C03569=1015.832,-110.510,-100.414,164.984,56.890,160.011
C03570=1015.836,-110.261,-100.421,164.987,56.884,160.010
C03571=1015.842,-110.011,-100.428,164.990,56.879,160.010
C03572=1015.846,-109.761,-100.435,164.993,56.872,160.010
C03573=1015.852,-109.511,-100.444,164.995,56.866,160.009
C03574=1015.857,-109.261,-100.452,164.999,56.860,160.009
C03575=1015.861,-109.012,-100.460,165.001,56.854,160.009
C03576=1015.866,-108.762,-100.468,165.003,56.847,160.008
C03577=1015.871,-108.511,-100.475,165.007,56.841,160.008
C03578=1015.876,-108.262,-100.484,165.010,56.835,160.007
C03579=1015.881,-108.012,-100.491,165.013,56.829,160.007
C03580=1015.886,-107.762,-100.499,165.016,56.823,160.007
C03581=1015.890,-107.513,-100.507,165.018,56.817,160.006
C03582=1015.895,-107.262,-100.515,165.022,56.811,160.006
C03583=1015.901,-107.013,-100.523,165.024,56.805,160.006
C03584=1015.905,-106.763,-100.531,165.027,56.799,160.005
C03585=1015.910,-106.513,-100.539,165.030,56.793,160.005
C03586=1015.915,-106.263,-100.547,165.033,56.787,160.005
C03587=1015.920,-106.014,-100.555,165.036,56.780,160.004
C03588=1015.925,-105.764,-100.563,165.039,56.774,160.004
C03589=1015.930,-105.514,-100.571,165.041,56.769,160.003
C03590=1015.934,-105.264,-100.579,165.045,56.762,160.003
C03591=1015.940,-105.014,-100.587,165.047,56.757,160.003
C03592=1015.945,-104.765,-100.596,165.051,56.750,160.003
C03593=1015.950,-104.514,-100.604,165.053,56.744,160.002
C03594=1015.955,-104.265,-100.612,165.056,56.738,160.002
C03595=1015.959,-104.015,-100.619,165.059,56.732,160.001
C03596=1015.965,-103.765,-100.628,165.062,56.726,160.001
C03597=1015.970,-103.515,-100.636,165.066,56.720,160.001
C03598=1015.974,-103.266,-100.644,165.068,56.713,160.000
C03599=1015.979,-103.016,-100.653,165.070,56.708,160.000
C03600=1015.984,-102.766,-100.661,165.074,56.701,160.000
C03601=1015.989,-102.516,-100.669,165.077,56.696,159.999
C03602=1015.995,-102.234,-100.678,165.080,56.689,159.999
C03603=1016.000,-101.952,-100.688,165.083,56.682,159.998
C03604=1016.006,-101.669,-100.697,165.087,56.674,159.998
C03605=1016.011,-101.387,-100.706,165.090,56.667,159.998
C03606=1016.016,-101.138,-100.715,165.093,56.662,159.997
C03607=1016.021,-100.887,-100.722,165.096,56.655,159.997
C03608=1016.027,-100.638,-100.731,165.098,56.649,159.996
C03609=1016.032,-100.388,-100.739,165.102,56.643,159.996
C03610=1016.037,-100.139,-100.747,165.104,56.636,159.996
C03611=1016.042,-99.888,-100.755,165.107,56.630,159.995
C03612=1016.046,-99.638,-100.764,165.110,56.624,159.995
C03613=1016.051,-99.389,-100.773,165.112,56.618,159.994
C03614=1016.057,-99.139,-100.781,165.116,56.612,159.994
C03615=1016.062,-98.889,-100.789,165.119,56.606,159.994
C03616=1016.066,-98.640,-100.797,165.122,56.599,159.993
C03617=1016.071,-98.390,-100.806,165.124,56.593,159.993
C03618=1016.077,-98.140,-100.814,165.128,56.587,159.993
C03619=1016.082,-97.890,-100.822,165.130,56.580,159.992
C03620=1016.086,-97.640,-100.831,165.134,56.574,159.992
C03621=1016.091,-97.390,-100.839,165.136,56.569,159.991
C03622=1016.096,-97.140,-100.849,165.139,56.563,159.991
C03623=1016.101,-96.890,-100.857,165.143,56.557,159.991
C03624=1016.107,-96.641,-100.865,165.145,56.551,159.990
C03625=1016.111,-96.391,-100.875,165.147,56.544,159.990
C03626=1016.116,-96.141,-100.883,165.151,56.538,159.990
C03627=1016.120,-95.892,-100.892,165.154,56.532,159.989
C03628=1016.126,-95.642,-100.900,165.157,56.526,159.989
C03629=1016.131,-95.392,-100.909,165.160,56.520,159.989
C03630=1016.135,-95.142,-100.918,165.162,56.514,159.988
C03631=1016.141,-94.892,-100.926,165.166,56.508,159.988
C03632=1016.146,-94.643,-100.935,165.168,56.502,159.987
C03633=1016.150,-94.393,-100.944,165.172,56.496,159.987
C03634=1016.156,-94.143,-100.952,165.174,56.489,159.987
C03635=1016.160,-93.893,-100.961,165.177,56.484,159.986
C03636=1016.165,-93.643,-100.970,165.180,56.477,159.986
C03637=1016.171,-93.394,-100.978,165.183,56.472,159.986
C03638=1016.175,-93.144,-100.987,165.186,56.465,159.985
C03639=1016.180,-92.894,-100.996,165.189,56.459,159.985
C03640=1016.185,-92.644,-101.005,165.192,56.453,159.985
C03641=1016.190,-92.394,-101.014,165.194,56.446,159.984
C03642=1016.196,-92.144,-101.022,165.197,56.441,159.983
C03643=1016.200,-91.894,-101.031,165.201,56.434,159.983
C03644=1016.206,-91.645,-101.040,165.203,56.428,159.983
C03645=1016.210,-91.395,-101.049,165.206,56.422,159.982
C03646=1016.215,-91.145,-101.058,165.209,56.416,159.982
C03647=1016.221,-90.896,-101.066,165.212,56.409,159.982
C03648=1016.225,-90.646,-101.075,165.215,56.403,159.981
C03649=1016.230,-90.396,-101.084,165.218,56.397,159.981
C03650=1016.235,-90.146,-101.093,165.221,56.391,159.980
C03651=1016.240,-89.896,-101.101,165.224,56.385,159.980
C03652=1016.246,-89.647,-101.111,165.227,56.379,159.980
C03653=1016.250,-89.397,-101.120,165.230,56.372,159.979
C03654=1016.256,-89.147,-101.128,165.233,56.366,159.979
C03655=1016.260,-88.897,-101.137,165.236,56.359,159.978
C03656=1016.266,-88.647,-101.146,165.238,56.354,159.978
C03657=1016.272,-88.398,-101.155,165.242,56.347,159.978
C03658=1016.276,-88.148,-101.164,165.244,56.341,159.977
C03659=1016.281,-87.898,-101.173,165.248,56.335,159.977
C03660=1016.286,-87.648,-101.182,165.250,56.328,159.976
C03661=1016.291,-87.398,-101.191,165.254,56.322,159.976
C03662=1016.296,-87.149,-101.200,165.256,56.316,159.975
C03663=1016.301,-86.899,-101.209,165.259,56.309,159.975
C03664=1016.307,-86.650,-101.217,165.261,56.303,159.975
C03665=1016.312,-86.399,-101.227,165.265,56.297,159.974
C03666=1016.317,-86.120,-101.237,165.268,56.290,159.974
C03667=1016.324,-85.839,-101.247,165.271,56.283,159.973
C03668=1016.329,-85.559,-101.257,165.274,56.275,159.973
C03669=1016.334,-85.278,-101.267,165.278,56.268,159.972
C03670=1016.340,-85.029,-101.276,165.281,56.262,159.972
C03671=1016.345,-84.779,-101.286,165.284,56.256,159.972
C03672=1016.350,-84.530,-101.294,165.287,56.250,159.971
C03673=1016.355,-84.280,-101.303,165.290,56.243,159.971
C03674=1016.361,-84.030,-101.313,165.293,56.237,159.970
C03675=1016.366,-83.780,-101.321,165.296,56.230,159.970
C03676=1016.370,-83.530,-101.330,165.298,56.224,159.969
C03677=1016.376,-83.281,-101.339,165.301,56.218,159.969
C03678=1016.381,-83.031,-101.348,165.305,56.211,159.969
C03679=1016.386,-82.780,-101.357,165.307,56.205,159.968
C03680=1016.392,-82.531,-101.367,165.310,56.198,159.968
C03681=1016.396,-82.281,-101.376,165.313,56.193,159.967
C03682=1016.402,-82.032,-101.385,165.316,56.186,159.967
C03683=1016.407,-81.782,-101.394,165.319,56.179,159.966
C03684=1016.412,-81.532,-101.403,165.322,56.173,159.966
C03685=1016.417,-81.282,-101.413,165.325,56.166,159.965
C03686=1016.422,-81.033,-101.421,165.328,56.160,159.965
C03687=1016.429,-80.783,-101.431,165.331,56.154,159.965
C03688=1016.433,-80.533,-101.440,165.334,56.147,159.964
C03689=1016.438,-80.283,-101.448,165.337,56.141,159.964
C03690=1016.443,-80.034,-101.458,165.340,56.134,159.963
C03691=1016.449,-79.784,-101.468,165.343,56.128,159.963
C03692=1016.454,-79.534,-101.477,165.346,56.122,159.962
C03693=1016.459,-79.285,-101.486,165.348,56.116,159.962
C03694=1016.464,-79.034,-101.496,165.352,56.109,159.962
C03695=1016.469,-78.784,-101.506,165.354,56.103,159.961
C03696=1016.474,-78.535,-101.515,165.357,56.096,159.961
C03697=1016.479,-78.285,-101.524,165.360,56.091,159.960
C03698=1016.484,-78.035,-101.534,165.364,56.085,159.960
C03699=1016.490,-77.786,-101.543,165.366,56.078,159.959
C03700=1016.494,-77.536,-101.552,165.370,56.072,159.959
C03701=1016.500,-77.286,-101.563,165.372,56.066,159.959
C03702=1016.505,-77.037,-101.572,165.375,56.059,159.958
C03703=1016.510,-76.787,-101.581,165.378,56.053,159.958
C03704=1016.515,-76.537,-101.591,165.381,56.046,159.957
C03705=1016.520,-76.287,-101.601,165.383,56.040,159.957
C03706=1016.525,-76.038,-101.609,165.387,56.034,159.956
C03707=1016.531,-75.787,-101.619,165.389,56.028,159.956
C03708=1016.536,-75.538,-101.629,165.392,56.021,159.955
C03709=1016.541,-75.287,-101.639,165.395,56.015,159.955
C03710=1016.546,-75.038,-101.648,165.398,56.008,159.955
C03711=1016.551,-74.789,-101.658,165.401,56.003,159.954
C03712=1016.557,-74.539,-101.668,165.404,55.996,159.954
C03713=1016.561,-74.289,-101.677,165.407,55.990,159.953
C03714=1016.567,-74.039,-101.687,165.410,55.983,159.953
C03715=1016.571,-73.789,-101.697,165.413,55.978,159.952
C03716=1016.576,-73.540,-101.707,165.416,55.972,159.952
C03717=1016.582,-73.290,-101.717,165.418,55.965,159.952
C03718=1016.587,-73.040,-101.727,165.421,55.959,159.951
C03719=1016.592,-72.790,-101.737,165.424,55.953,159.951
C03720=1016.597,-72.541,-101.747,165.427,55.947,159.950
C03721=1016.602,-72.291,-101.757,165.431,55.941,159.950
C03722=1016.607,-72.041,-101.767,165.433,55.934,159.949
C03723=1016.612,-71.792,-101.776,165.436,55.929,159.949
C03724=1016.617,-71.542,-101.787,165.439,55.922,159.949
C03725=1016.622,-71.292,-101.796,165.441,55.916,159.948
C03726=1016.628,-71.042,-101.806,165.445,55.910,159.948
C03727=1016.632,-70.793,-101.816,165.447,55.904,159.947
C03728=1016.638,-70.543,-101.826,165.451,55.897,159.947
C03729=1016.643,-70.293,-101.836,165.453,55.891,159.946
C03730=1016.649,-70.015,-101.847,165.456,55.884,159.946
C03731=1016.654,-69.737,-101.859,165.460,55.877,159.945
C03732=1016.660,-69.458,-101.870,165.463,55.870,159.945
C03733=1016.665,-69.180,-101.880,165.466,55.864,159.944
C03734=1016.671,-68.930,-101.890,165.469,55.857,159.944
C03735=1016.676,-68.681,-101.900,165.472,55.851,159.944
C03736=1016.681,-68.430,-101.910,165.475,55.844,159.943
C03737=1016.686,-68.181,-101.920,165.478,55.839,159.943
C03738=1016.692,-67.932,-101.931,165.481,55.832,159.942
C03739=1016.697,-67.681,-101.941,165.484,55.826,159.942
C03740=1016.702,-67.432,-101.951,165.487,55.819,159.941
C03741=1016.707,-67.182,-101.961,165.489,55.814,159.941
C03742=1016.712,-66.933,-101.971,165.493,55.807,159.941
C03743=1016.717,-66.682,-101.982,165.495,55.801,159.940
C03744=1016.722,-66.433,-101.992,165.499,55.794,159.940
C03745=1016.727,-66.183,-102.002,165.501,55.788,159.939
C03746=1016.732,-65.933,-102.012,165.504,55.782,159.939
C03747=1016.738,-65.684,-102.022,165.507,55.775,159.938
C03748=1016.743,-65.434,-102.033,165.510,55.769,159.938
C03749=1016.748,-65.184,-102.042,165.512,55.763,159.937
C03750=1016.753,-64.934,-102.053,165.516,55.756,159.937
C03751=1016.758,-64.685,-102.062,165.518,55.750,159.936
C03752=1016.764,-64.435,-102.072,165.522,55.744,159.936
C03753=1016.769,-64.185,-102.083,165.524,55.738,159.935
C03754=1016.774,-63.936,-102.093,165.527,55.731,159.935
C03755=1016.780,-63.686,-102.103,165.530,55.725,159.934
C03756=1016.784,-63.436,-102.113,165.533,55.719,159.934
C03757=1016.790,-63.186,-102.123,165.537,55.712,159.934
C03758=1016.796,-62.937,-102.134,165.539,55.705,159.933
C03759=1016.800,-62.687,-102.144,165.543,55.699,159.933
C03760=1016.806,-62.437,-102.154,165.545,55.693,159.932
C03761=1016.811,-62.187,-102.164,165.548,55.686,159.932
C03762=1016.816,-61.938,-102.175,165.551,55.680,159.931
C03763=1016.822,-61.688,-102.185,165.554,55.674,159.931
C03764=1016.827,-61.438,-102.195,165.556,55.667,159.930
C03765=1016.831,-61.188,-102.205,165.560,55.661,159.930
C03766=1016.837,-60.939,-102.216,165.562,55.655,159.929
C03767=1016.843,-60.689,-102.227,165.565,55.648,159.929
C03768=1016.847,-60.439,-102.236,165.568,55.641,159.928
C03769=1016.853,-60.190,-102.247,165.571,55.635,159.928
C03770=1016.859,-59.940,-102.257,165.574,55.629,159.927
C03771=1016.863,-59.690,-102.267,165.576,55.622,159.927
C03772=1016.869,-59.440,-102.277,165.580,55.615,159.926
C03773=1016.875,-59.191,-102.288,165.582,55.610,159.926
C03774=1016.880,-58.940,-102.298,165.586,55.603,159.925
C03775=1016.885,-58.691,-102.308,165.589,55.596,159.925
C03776=1016.891,-58.442,-102.319,165.591,55.590,159.924
C03777=1016.896,-58.191,-102.329,165.595,55.584,159.924
C03778=1016.902,-57.942,-102.340,165.597,55.577,159.923
C03779=1016.907,-57.693,-102.350,165.600,55.570,159.923
C03780=1016.912,-57.442,-102.360,165.603,55.564,159.922
C03781=1016.918,-57.193,-102.371,165.606,55.557,159.922
C03782=1016.922,-56.943,-102.382,165.609,55.550,159.921
C03783=1016.928,-56.694,-102.392,165.612,55.545,159.921
C03784=1016.933,-56.444,-102.402,165.615,55.538,159.920
C03785=1016.938,-56.194,-102.412,165.618,55.531,159.920
C03786=1016.944,-55.944,-102.423,165.620,55.525,159.919
C03787=1016.950,-55.694,-102.434,165.623,55.518,159.919
C03788=1016.955,-55.445,-102.444,165.626,55.512,159.918
C03789=1016.960,-55.195,-102.454,165.629,55.506,159.918
C03790=1016.966,-54.946,-102.465,165.633,55.499,159.917
C03791=1016.971,-54.695,-102.475,165.635,55.492,159.917
C03792=1016.977,-54.445,-102.485,165.638,55.486,159.916
C03793=1016.982,-54.197,-102.496,165.640,55.479,159.915
C03794=1016.988,-53.919,-102.508,165.644,55.471,159.915
C03795=1016.995,-53.642,-102.520,165.647,55.465,159.914
C03796=1017.000,-53.365,-102.531,165.650,55.457,159.914
C03797=1017.006,-53.088,-102.543,165.654,55.450,159.913
C03798=1017.012,-52.838,-102.553,165.657,55.444,159.913
C03799=1017.017,-52.588,-102.564,165.660,55.437,159.912
C03800=1017.022,-52.338,-102.575,165.662,55.430,159.912
C03801=1017.027,-52.089,-102.585,165.665,55.424,159.911
C03802=1017.033,-51.839,-102.596,165.668,55.417,159.911
C03803=1017.038,-51.589,-102.606,165.671,55.410,159.910
C03804=1017.044,-51.340,-102.617,165.674,55.404,159.909
C03805=1017.050,-51.090,-102.627,165.677,55.397,159.909
C03806=1017.055,-50.840,-102.638,165.679,55.391,159.908
///RCONF 1,0,0,0,0,0,0,0,0,0,0,0,0,0,0,0,0,0,0,0,0,0,0,0
C03807=1017.060,-50.590,-102.649,165.683,55.384,159.908
C03808=1017.065,-50.340,-102.661,165.685,55.378,159.907
C03809=1017.071,-50.090,-102.671,165.689,55.371,159.907
C03810=1017.076,-49.841,-102.682,165.691,55.366,159.906
C03811=1017.081,-49.591,-102.693,165.695,55.359,159.906
C03812=1017.086,-49.341,-102.705,165.697,55.353,159.905
C03813=1017.092,-49.091,-102.715,165.701,55.347,159.905
C03814=1017.097,-48.842,-102.725,165.703,55.340,159.904
C03815=1017.102,-48.593,-102.737,165.705,55.334,159.904
C03816=1017.108,-48.343,-102.748,165.708,55.327,159.903
C03817=1017.113,-48.093,-102.759,165.711,55.321,159.903
C03818=1017.119,-47.844,-102.770,165.714,55.315,159.902
C03819=1017.123,-47.593,-102.781,165.716,55.308,159.902
C03820=1017.129,-47.344,-102.792,165.720,55.302,159.901
C03821=1017.134,-47.094,-102.803,165.722,55.296,159.901
C03822=1017.140,-46.845,-102.814,165.726,55.289,159.900
C03823=1017.145,-46.595,-102.826,165.728,55.283,159.900
C03824=1017.150,-46.345,-102.837,165.731,55.276,159.899
C03825=1017.155,-46.095,-102.848,165.734,55.270,159.899
C03826=1017.161,-45.846,-102.859,165.737,55.264,159.898
C03827=1017.166,-45.596,-102.870,165.739,55.257,159.898
C03828=1017.172,-45.347,-102.881,165.743,55.251,159.897
C03829=1017.177,-45.096,-102.892,165.746,55.244,159.897
C03830=1017.182,-44.847,-102.903,165.749,55.238,159.896
C03831=1017.187,-44.597,-102.914,165.752,55.231,159.896
C03832=1017.193,-44.347,-102.925,165.754,55.225,159.895
C03833=1017.198,-44.098,-102.937,165.757,55.218,159.895
C03834=1017.204,-43.848,-102.948,165.760,55.212,159.894
C03835=1017.209,-43.598,-102.959,165.763,55.205,159.893
C03836=1017.215,-43.349,-102.970,165.765,55.199,159.893
C03837=1017.220,-43.099,-102.981,165.769,55.193,159.893
C03838=1017.225,-42.850,-102.992,165.771,55.186,159.892
C03839=1017.230,-42.600,-103.004,165.775,55.180,159.891
C03840=1017.236,-42.350,-103.015,165.777,55.173,159.891
C03841=1017.241,-42.101,-103.026,165.780,55.167,159.890
C03842=1017.247,-41.850,-103.037,165.782,55.160,159.890
C03843=1017.252,-41.601,-103.049,165.786,55.154,159.889
C03844=1017.258,-41.351,-103.060,165.789,55.147,159.889
C03845=1017.263,-41.101,-103.071,165.791,55.140,159.888
C03846=1017.269,-40.852,-103.082,165.794,55.134,159.887
C03847=1017.274,-40.602,-103.093,165.797,55.128,159.887
C03848=1017.280,-40.352,-103.104,165.800,55.121,159.887
C03849=1017.285,-40.103,-103.116,165.803,55.115,159.886
C03850=1017.291,-39.854,-103.127,165.806,55.108,159.885
C03851=1017.296,-39.604,-103.139,165.809,55.102,159.885
C03852=1017.301,-39.353,-103.151,165.811,55.095,159.884
C03853=1017.307,-39.104,-103.162,165.815,55.088,159.884
C03854=1017.312,-38.854,-103.173,165.817,55.082,159.883
C03855=1017.317,-38.604,-103.185,165.820,55.077,159.883
C03856=1017.322,-38.355,-103.197,165.823,55.070,159.882
C03857=1017.328,-38.106,-103.208,165.825,55.063,159.881
C03858=1017.334,-37.828,-103.221,165.829,55.057,159.881
C03859=1017.339,-37.551,-103.233,165.831,55.049,159.880
C03860=1017.346,-37.275,-103.246,165.835,55.043,159.880
C03861=1017.351,-36.998,-103.259,165.838,55.035,159.879
C03862=1017.356,-36.748,-103.270,165.841,55.028,159.879
C03863=1017.362,-36.499,-103.283,165.843,55.023,159.878
C03864=1017.368,-36.249,-103.294,165.847,55.016,159.878
C03865=1017.373,-35.999,-103.305,165.849,55.010,159.877
C03866=1017.378,-35.750,-103.318,165.852,55.003,159.876
C03867=1017.383,-35.500,-103.329,165.855,54.997,159.876
C03868=1017.389,-35.250,-103.341,165.858,54.990,159.875
C03869=1017.395,-35.001,-103.352,165.860,54.984,159.875
C03870=1017.400,-34.751,-103.364,165.864,54.978,159.874
C03871=1017.405,-34.501,-103.375,165.866,54.971,159.874
C03872=1017.410,-34.252,-103.388,165.870,54.965,159.873
C03873=1017.416,-34.002,-103.399,165.872,54.958,159.873
C03874=1017.422,-33.752,-103.410,165.875,54.952,159.872
C03875=1017.427,-33.503,-103.422,165.877,54.945,159.871
C03876=1017.432,-33.253,-103.434,165.881,54.939,159.871
C03877=1017.438,-33.003,-103.446,165.883,54.932,159.870
C03878=1017.443,-32.753,-103.458,165.886,54.925,159.870
C03879=1017.449,-32.504,-103.469,165.888,54.919,159.869
C03880=1017.454,-32.255,-103.481,165.892,54.912,159.869
C03881=1017.459,-32.004,-103.493,165.895,54.907,159.868
C03882=1017.465,-31.755,-103.505,165.898,54.900,159.868
C03883=1017.470,-31.505,-103.517,165.900,54.894,159.867
C03884=1017.476,-31.256,-103.528,165.903,54.887,159.867
C03885=1017.481,-31.006,-103.540,165.906,54.881,159.866
C03886=1017.486,-30.756,-103.551,165.909,54.874,159.865
C03887=1017.492,-30.507,-103.564,165.911,54.868,159.865
C03888=1017.497,-30.256,-103.575,165.915,54.861,159.864
C03889=1017.503,-30.008,-103.587,165.917,54.855,159.864
C03890=1017.508,-29.758,-103.599,165.920,54.848,159.863
C03891=1017.514,-29.508,-103.611,165.923,54.842,159.862
C03892=1017.519,-29.258,-103.623,165.926,54.835,159.862
C03893=1017.525,-29.009,-103.635,165.928,54.829,159.861
C03894=1017.531,-28.759,-103.646,165.931,54.822,159.861
C03895=1017.536,-28.510,-103.658,165.935,54.815,159.860
C03896=1017.541,-28.260,-103.670,165.937,54.809,159.860
C03897=1017.547,-28.010,-103.682,165.940,54.802,159.859
C03898=1017.552,-27.760,-103.694,165.942,54.795,159.858
C03899=1017.557,-27.511,-103.706,165.946,54.789,159.858
C03900=1017.563,-27.261,-103.718,165.948,54.783,159.857
C03901=1017.568,-27.011,-103.730,165.951,54.777,159.857
C03902=1017.574,-26.762,-103.742,165.954,54.770,159.856
C03903=1017.580,-26.512,-103.755,165.956,54.764,159.855
C03904=1017.585,-26.262,-103.766,165.959,54.757,159.855
C03905=1017.591,-26.012,-103.779,165.962,54.751,159.854
C03906=1017.596,-25.763,-103.791,165.965,54.744,159.854
C03907=1017.601,-25.514,-103.803,165.968,54.739,159.853
C03908=1017.607,-25.264,-103.815,165.970,54.732,159.853
C03909=1017.611,-25.014,-103.828,165.973,54.726,159.852
C03910=1017.617,-24.764,-103.840,165.976,54.719,159.852
C03911=1017.623,-24.515,-103.852,165.979,54.713,159.851
C03912=1017.628,-24.265,-103.864,165.981,54.706,159.850
C03913=1017.633,-24.015,-103.876,165.985,54.700,159.850
C03914=1017.639,-23.766,-103.889,165.987,54.693,159.849
C03915=1017.645,-23.516,-103.901,165.989,54.687,159.849
C03916=1017.650,-23.266,-103.913,165.993,54.680,159.848
C03917=1017.655,-23.017,-103.925,165.995,54.674,159.847
C03918=1017.661,-22.767,-103.937,165.998,54.667,159.847
C03919=1017.666,-22.518,-103.950,166.001,54.661,159.846
C03920=1017.671,-22.268,-103.963,166.004,54.654,159.846
C03921=1017.676,-22.018,-103.974,166.006,54.648,159.845
C03922=1017.683,-21.741,-103.988,166.010,54.641,159.845
C03923=1017.689,-21.463,-104.001,166.012,54.634,159.844
C03924=1017.695,-21.185,-104.015,166.015,54.627,159.843
C03925=1017.701,-20.907,-104.029,166.019,54.620,159.843
C03926=1017.707,-20.658,-104.041,166.022,54.613,159.842
C03927=1017.713,-20.408,-104.054,166.024,54.606,159.841
C03928=1017.718,-20.158,-104.065,166.027,54.600,159.841
C03929=1017.724,-19.908,-104.078,166.029,54.593,159.840
C03930=1017.728,-19.659,-104.091,166.033,54.587,159.840
C03931=1017.734,-19.409,-104.103,166.035,54.580,159.839
C03932=1017.739,-19.160,-104.116,166.038,54.574,159.838
C03933=1017.745,-18.910,-104.128,166.041,54.567,159.838
C03934=1017.751,-18.661,-104.140,166.044,54.561,159.837
C03935=1017.756,-18.411,-104.153,166.046,54.555,159.837
C03936=1017.762,-18.162,-104.165,166.050,54.548,159.836
C03937=1017.768,-17.912,-104.178,166.052,54.542,159.835
C03938=1017.773,-17.663,-104.190,166.055,54.535,159.835
C03939=1017.778,-17.412,-104.202,166.058,54.529,159.834
C03940=1017.783,-17.163,-104.214,166.061,54.522,159.834
C03941=1017.789,-16.913,-104.227,166.063,54.515,159.833
C03942=1017.795,-16.663,-104.240,166.066,54.508,159.832
C03943=1017.800,-16.414,-104.252,166.069,54.502,159.832
C03944=1017.806,-16.164,-104.264,166.072,54.495,159.831
C03945=1017.811,-15.915,-104.276,166.074,54.489,159.830
C03946=1017.817,-15.665,-104.290,166.078,54.482,159.830
C03947=1017.822,-15.416,-104.302,166.080,54.476,159.829
C03948=1017.828,-15.166,-104.315,166.082,54.470,159.829
C03949=1017.833,-14.917,-104.328,166.086,54.463,159.828
C03950=1017.839,-14.667,-104.340,166.088,54.457,159.827
C03951=1017.844,-14.417,-104.354,166.090,54.451,159.827
C03952=1017.849,-14.167,-104.366,166.094,54.444,159.826
C03953=1017.855,-13.917,-104.378,166.096,54.438,159.826
C03954=1017.860,-13.669,-104.392,166.099,54.431,159.825
C03955=1017.866,-13.419,-104.404,166.102,54.425,159.824
C03956=1017.871,-13.168,-104.417,166.104,54.419,159.824
C03957=1017.876,-12.919,-104.430,166.107,54.412,159.823
C03958=1017.882,-12.669,-104.442,166.110,54.406,159.823
C03959=1017.888,-12.420,-104.456,166.113,54.399,159.822
C03960=1017.893,-12.171,-104.468,166.115,54.393,159.821
C03961=1017.898,-11.920,-104.481,166.118,54.387,159.821
C03962=1017.903,-11.671,-104.494,166.121,54.380,159.820
C03963=1017.909,-11.421,-104.506,166.123,54.374,159.820
C03964=1017.915,-11.172,-104.520,166.127,54.367,159.819
C03965=1017.920,-10.923,-104.532,166.129,54.361,159.818
C03966=1017.926,-10.673,-104.545,166.132,54.355,159.818
C03967=1017.931,-10.423,-104.558,166.135,54.348,159.817
C03968=1017.937,-10.174,-104.571,166.137,54.342,159.817
C03969=1017.942,-9.924,-104.584,166.141,54.335,159.816
C03970=1017.948,-9.674,-104.597,166.143,54.329,159.815
C03971=1017.954,-9.425,-104.609,166.146,54.321,159.815
C03972=1017.959,-9.175,-104.623,166.148,54.315,159.814
C03973=1017.965,-8.925,-104.635,166.151,54.309,159.813
C03974=1017.969,-8.676,-104.648,166.154,54.302,159.813
C03975=1017.975,-8.427,-104.661,166.156,54.296,159.812
C03976=1017.981,-8.177,-104.674,166.160,54.289,159.812
C03977=1017.986,-7.926,-104.687,166.162,54.283,159.811
C03978=1017.992,-7.678,-104.700,166.165,54.277,159.811
C03979=1017.997,-7.428,-104.713,166.167,54.270,159.810
C03980=1018.003,-7.178,-104.725,166.171,54.263,159.809
C03981=1018.009,-6.929,-104.738,166.173,54.257,159.808
C03982=1018.014,-6.679,-104.752,166.175,54.251,159.808
C03983=1018.020,-6.429,-104.764,166.179,54.244,159.807
C03984=1018.025,-6.180,-104.778,166.181,54.238,159.807
C03985=1018.031,-5.930,-104.790,166.184,54.230,159.806
C03986=1018.038,-5.650,-104.805,166.187,54.223,159.805
C03987=1018.043,-5.371,-104.820,166.190,54.216,159.804
C03988=1018.050,-5.091,-104.834,166.193,54.209,159.804
C03989=1018.056,-4.812,-104.849,166.196,54.202,159.803
C03990=1018.062,-4.562,-104.862,166.199,54.194,159.802
C03991=1018.067,-4.313,-104.875,166.201,54.188,159.802
C03992=1018.072,-4.063,-104.888,166.204,54.182,159.801
C03993=1018.078,-3.813,-104.902,166.207,54.175,159.801
C03994=1018.083,-3.563,-104.915,166.210,54.169,159.800
C03995=1018.089,-3.314,-104.928,166.212,54.163,159.799
C03996=1018.094,-3.064,-104.941,166.215,54.156,159.799
C03997=1018.099,-2.815,-104.955,166.218,54.150,159.798
C03998=1018.105,-2.565,-104.969,166.220,54.144,159.797
C03999=1018.111,-2.315,-104.981,166.223,54.137,159.797
C04000=1018.116,-2.066,-104.995,166.226,54.131,159.796
C04001=1018.121,-1.817,-105.009,166.228,54.125,159.796
C04002=1018.126,-1.567,-105.022,166.232,54.118,159.795
C04003=1018.132,-1.317,-105.036,166.234,54.112,159.794
C04004=1018.138,-1.068,-105.049,166.236,54.106,159.794
C04005=1018.143,-0.818,-105.062,166.239,54.099,159.793
C04006=1018.148,-0.569,-105.076,166.242,54.093,159.793
C04007=1018.153,-0.319,-105.089,166.244,54.087,159.792
C04008=1018.159,-0.069,-105.102,166.247,54.080,159.791
C04009=1018.165,0.180,-105.116,166.250,54.074,159.791
C04010=1018.170,0.430,-105.130,166.253,54.068,159.790
C04011=1018.175,0.680,-105.143,166.255,54.061,159.789
C04012=1018.180,0.929,-105.156,166.258,54.055,159.789
C04013=1018.186,1.178,-105.170,166.261,54.049,159.788
C04014=1018.192,1.428,-105.183,166.263,54.042,159.788
C04015=1018.197,1.678,-105.197,166.266,54.035,159.787
C04016=1018.203,1.927,-105.211,166.268,54.029,159.786
C04017=1018.209,2.177,-105.224,166.272,54.022,159.786
C04018=1018.214,2.426,-105.238,166.274,54.016,159.785
C04019=1018.219,2.676,-105.251,166.277,54.010,159.784
C04020=1018.224,2.925,-105.264,166.280,54.003,159.784
C04021=1018.230,3.175,-105.278,166.282,53.997,159.783
C04022=1018.236,3.424,-105.291,166.285,53.991,159.783
C04023=1018.241,3.674,-105.305,166.288,53.983,159.782
C04024=1018.247,3.924,-105.318,166.290,53.977,159.781
C04025=1018.252,4.174,-105.332,166.292,53.971,159.780
C04026=1018.258,4.423,-105.346,166.296,53.964,159.780
C04027=1018.264,4.672,-105.359,166.298,53.958,159.779
C04028=1018.269,4.922,-105.373,166.301,53.952,159.779
C04029=1018.274,5.172,-105.386,166.304,53.945,159.778
C04030=1018.280,5.422,-105.400,166.306,53.939,159.777
C04031=1018.286,5.671,-105.414,166.309,53.932,159.777
C04032=1018.292,5.921,-105.427,166.312,53.926,159.776
C04033=1018.297,6.169,-105.441,166.314,53.920,159.775
C04034=1018.302,6.419,-105.455,166.317,53.912,159.775
C04035=1018.307,6.669,-105.468,166.320,53.906,159.774
C04036=1018.313,6.918,-105.481,166.322,53.900,159.773
C04037=1018.319,7.168,-105.495,166.325,53.893,159.773
C04038=1018.324,7.418,-105.509,166.327,53.886,159.772
C04039=1018.330,7.667,-105.523,166.331,53.880,159.771
C04040=1018.335,7.917,-105.537,166.333,53.874,159.771
C04041=1018.342,8.166,-105.550,166.336,53.867,159.770
C04042=1018.347,8.416,-105.564,166.339,53.860,159.769
C04043=1018.352,8.665,-105.578,166.341,53.854,159.769
C04044=1018.358,8.915,-105.592,166.344,53.847,159.768
C04045=1018.363,9.165,-105.605,166.347,53.841,159.767
C04046=1018.369,9.414,-105.618,166.349,53.834,159.767
C04047=1018.375,9.664,-105.632,166.352,53.828,159.766
C04048=1018.380,9.913,-105.646,166.355,53.821,159.765
C04049=1018.386,10.163,-105.660,166.358,53.814,159.765
C04050=1018.393,10.444,-105.675,166.361,53.807,159.764
C04051=1018.399,10.726,-105.691,166.363,53.800,159.763
C04052=1018.405,11.008,-105.706,166.366,53.792,159.762
C04053=1018.411,11.289,-105.722,166.369,53.785,159.762
C04054=1018.418,11.538,-105.736,166.371,53.778,159.761
C04055=1018.423,11.788,-105.749,166.375,53.772,159.760
C04056=1018.429,12.038,-105.763,166.377,53.765,159.760
C04057=1018.434,12.287,-105.777,166.380,53.758,159.759
C04058=1018.440,12.550,-105.791,166.383,53.752,159.758
C04059=1018.446,12.813,-105.806,166.386,53.745,159.757
C04060=1018.452,13.076,-105.820,166.389,53.737,159.757
C04061=1018.458,13.339,-105.835,166.391,53.731,159.756
C04062=1018.463,13.588,-105.849,166.394,53.724,159.755
C04063=1018.469,13.838,-105.863,166.396,53.718,159.755
C04064=1018.474,14.087,-105.878,166.399,53.712,159.754
C04065=1018.480,14.336,-105.891,166.402,53.705,159.753
C04066=1018.485,14.586,-105.905,166.405,53.699,159.753
C04067=1018.491,14.836,-105.919,166.407,53.692,159.752
C04068=1018.496,15.085,-105.933,166.410,53.685,159.751
C04069=1018.502,15.335,-105.949,166.413,53.679,159.751
C04070=1018.508,15.585,-105.962,166.415,53.673,159.750
C04071=1018.513,15.834,-105.976,166.418,53.666,159.749
C04072=1018.518,16.084,-105.990,166.420,53.660,159.749
C04073=1018.524,16.333,-106.005,166.423,53.654,159.748
C04074=1018.530,16.582,-106.019,166.425,53.647,159.747
C04075=1018.535,16.832,-106.032,166.428,53.640,159.746
C04076=1018.541,17.082,-106.046,166.431,53.634,159.746
C04077=1018.546,17.331,-106.061,166.433,53.628,159.745
C04078=1018.553,17.581,-106.075,166.437,53.621,159.745
C04079=1018.557,17.831,-106.090,166.439,53.614,159.744
C04080=1018.563,18.080,-106.103,166.441,53.608,159.743
C04081=1018.569,18.329,-106.118,166.444,53.602,159.743
C04082=1018.574,18.579,-106.132,166.446,53.595,159.742
C04083=1018.579,18.828,-106.146,166.450,53.588,159.741
C04084=1018.586,19.078,-106.161,166.452,53.582,159.741
C04085=1018.591,19.328,-106.175,166.455,53.576,159.740
C04086=1018.596,19.578,-106.189,166.457,53.569,159.739
C04087=1018.602,19.826,-106.204,166.460,53.562,159.738
C04088=1018.607,20.076,-106.217,166.463,53.556,159.738
C04089=1018.613,20.325,-106.232,166.465,53.550,159.737
C04090=1018.618,20.576,-106.247,166.468,53.543,159.736
C04091=1018.624,20.825,-106.261,166.471,53.537,159.736
C04092=1018.630,21.074,-106.275,166.473,53.531,159.735
C04093=1018.635,21.324,-106.289,166.475,53.524,159.734
C04094=1018.640,21.573,-106.304,166.478,53.517,159.734
C04095=1018.646,21.823,-106.319,166.481,53.511,159.733
C04096=1018.652,22.072,-106.333,166.483,53.505,159.732
C04097=1018.658,22.322,-106.347,166.487,53.498,159.732
C04098=1018.662,22.572,-106.361,166.489,53.492,159.731
C04099=1018.668,22.821,-106.376,166.491,53.485,159.730
C04100=1018.674,23.071,-106.390,166.495,53.479,159.730
C04101=1018.680,23.320,-106.405,166.497,53.472,159.729
C04102=1018.685,23.570,-106.419,166.499,53.466,159.728
C04103=1018.690,23.819,-106.434,166.503,53.459,159.728
C04104=1018.697,24.069,-106.448,166.505,53.452,159.727
C04105=1018.702,24.318,-106.463,166.507,53.446,159.726
C04106=1018.707,24.568,-106.477,166.511,53.440,159.726
C04107=1018.713,24.817,-106.492,166.513,53.433,159.725
C04108=1018.719,25.067,-106.506,166.515,53.427,159.724
C04109=1018.724,25.316,-106.521,166.519,53.420,159.723
C04110=1018.729,25.566,-106.535,166.521,53.413,159.723
C04111=1018.735,25.815,-106.550,166.523,53.407,159.722
C04112=1018.742,26.064,-106.565,166.525,53.401,159.721
C04113=1018.746,26.314,-106.579,166.528,53.394,159.721
C04114=1018.752,26.584,-106.595,166.532,53.387,159.720
C04115=1018.759,26.854,-106.611,166.534,53.381,159.719
C04116=1018.765,27.123,-106.626,166.537,53.373,159.718
C04117=1018.771,27.394,-106.642,166.540,53.366,159.718
C04118=1018.776,27.643,-106.657,166.542,53.359,159.717
C04119=1018.782,27.892,-106.671,166.545,53.353,159.716
C04120=1018.787,28.143,-106.686,166.548,53.347,159.716
C04121=1018.793,28.392,-106.701,166.550,53.341,159.715
C04122=1018.798,28.641,-106.716,166.553,53.334,159.714
C04123=1018.804,28.891,-106.731,166.555,53.328,159.713
C04124=1018.809,29.140,-106.745,166.558,53.321,159.713
C04125=1018.815,29.389,-106.760,166.561,53.315,159.712
C04126=1018.820,29.639,-106.776,166.563,53.308,159.711
C04127=1018.826,29.888,-106.790,166.565,53.302,159.711
C04128=1018.831,30.138,-106.805,166.569,53.295,159.710
C04129=1018.837,30.388,-106.819,166.571,53.289,159.709
C04130=1018.842,30.637,-106.835,166.573,53.282,159.708
C04131=1018.848,30.886,-106.849,166.576,53.276,159.708
C04132=1018.853,31.137,-106.864,166.579,53.269,159.707
C04133=1018.859,31.386,-106.879,166.581,53.263,159.706
C04134=1018.864,31.635,-106.894,166.584,53.257,159.706
C04135=1018.871,31.885,-106.909,166.587,53.250,159.705
C04136=1018.876,32.134,-106.924,166.589,53.244,159.704
C04137=1018.881,32.383,-106.938,166.592,53.237,159.704
C04138=1018.887,32.633,-106.953,166.594,53.231,159.703
C04139=1018.893,32.882,-106.968,166.597,53.224,159.702
C04140=1018.898,33.132,-106.983,166.600,53.218,159.702
C04141=1018.903,33.382,-106.999,166.602,53.211,159.701
C04142=1018.909,33.631,-107.013,166.605,53.205,159.700
C04143=1018.914,33.881,-107.028,166.608,53.198,159.699
C04144=1018.920,34.130,-107.043,166.610,53.192,159.699
C04145=1018.925,34.379,-107.058,166.612,53.186,159.698
C04146=1018.932,34.629,-107.073,166.616,53.178,159.697
C04147=1018.937,34.878,-107.088,166.618,53.172,159.697
C04148=1018.943,35.128,-107.103,166.620,53.166,159.696
C04149=1018.948,35.378,-107.117,166.624,53.159,159.695
C04150=1018.954,35.627,-107.132,166.626,53.153,159.694
C04151=1018.959,35.877,-107.147,166.628,53.146,159.694
C04152=1018.965,36.126,-107.162,166.632,53.140,159.693
C04153=1018.971,36.376,-107.178,166.634,53.133,159.692
C04154=1018.976,36.625,-107.192,166.636,53.127,159.692
C04155=1018.982,36.875,-107.208,166.639,53.121,159.691
C04156=1018.987,37.124,-107.223,166.642,53.113,159.690
C04157=1018.993,37.374,-107.238,166.644,53.107,159.689
C04158=1018.998,37.623,-107.254,166.647,53.101,159.689
C04159=1019.004,37.873,-107.269,166.649,53.094,159.688
C04160=1019.009,38.122,-107.284,166.652,53.088,159.687
C04161=1019.014,38.371,-107.299,166.655,53.082,159.687
C04162=1019.020,38.621,-107.314,166.657,53.075,159.686
C04163=1019.026,38.870,-107.329,166.659,53.069,159.685
C04164=1019.031,39.120,-107.345,166.663,53.062,159.685
C04165=1019.036,39.369,-107.360,166.665,53.056,159.684
C04166=1019.042,39.619,-107.376,166.667,53.050,159.683
C04167=1019.048,39.868,-107.391,166.670,53.043,159.682
C04168=1019.054,40.118,-107.406,166.673,53.036,159.682
C04169=1019.059,40.367,-107.421,166.676,53.030,159.681
C04170=1019.064,40.617,-107.437,166.678,53.024,159.680
C04171=1019.070,40.866,-107.452,166.680,53.017,159.679
C04172=1019.076,41.116,-107.467,166.684,53.011,159.679
C04173=1019.081,41.365,-107.482,166.686,53.004,159.678
C04174=1019.087,41.615,-107.498,166.688,52.998,159.677
C04175=1019.092,41.864,-107.514,166.691,52.992,159.677
C04176=1019.098,42.113,-107.528,166.694,52.985,159.676
C04177=1019.103,42.363,-107.544,166.696,52.979,159.675
C04178=1019.109,42.646,-107.562,166.699,52.971,159.675
C04179=1019.115,42.929,-107.579,166.703,52.964,159.674
C04180=1019.122,43.212,-107.597,166.705,52.957,159.673
C04181=1019.128,43.495,-107.615,166.707,52.950,159.672
C04182=1019.133,43.744,-107.630,166.710,52.944,159.671
C04183=1019.139,43.994,-107.646,166.713,52.937,159.671
C04184=1019.144,44.243,-107.662,166.716,52.931,159.670
C04185=1019.150,44.493,-107.677,166.718,52.924,159.669
C04186=1019.155,44.742,-107.692,166.721,52.918,159.669
C04187=1019.161,44.992,-107.709,166.723,52.912,159.668
C04188=1019.166,45.241,-107.724,166.726,52.906,159.667
C04189=1019.171,45.491,-107.739,166.729,52.899,159.666
C04190=1019.177,45.740,-107.755,166.731,52.893,159.666
C04191=1019.182,45.990,-107.771,166.734,52.887,159.665
C04192=1019.188,46.239,-107.787,166.736,52.880,159.664
C04193=1019.192,46.488,-107.803,166.738,52.874,159.664
C04194=1019.198,46.738,-107.818,166.742,52.867,159.663
C04195=1019.203,46.987,-107.834,166.744,52.861,159.662
C04196=1019.209,47.237,-107.850,166.746,52.854,159.661
C04197=1019.214,47.486,-107.866,166.749,52.848,159.661
C04198=1019.220,47.736,-107.881,166.751,52.842,159.660
C04199=1019.226,47.986,-107.897,166.755,52.835,159.659
C04200=1019.231,48.234,-107.913,166.757,52.829,159.659
C04201=1019.237,48.484,-107.928,166.759,52.822,159.658
C04202=1019.242,48.733,-107.944,166.762,52.816,159.657
C04203=1019.248,48.983,-107.960,166.764,52.810,159.657
C04204=1019.254,49.232,-107.976,166.767,52.803,159.656
C04205=1019.259,49.481,-107.991,166.770,52.797,159.655
C04206=1019.264,49.731,-108.007,166.773,52.791,159.654
C04207=1019.269,49.980,-108.023,166.775,52.784,159.654
C04208=1019.275,50.230,-108.039,166.778,52.778,159.653
C04209=1019.281,50.480,-108.055,166.780,52.771,159.652
C04210=1019.286,50.729,-108.070,166.783,52.765,159.652
C04211=1019.292,50.978,-108.086,166.785,52.758,159.651
C04212=1019.297,51.228,-108.102,166.788,52.752,159.650
C04213=1019.303,51.477,-108.118,166.791,52.746,159.649
C04214=1019.308,51.727,-108.133,166.793,52.739,159.649
C04215=1019.314,51.976,-108.150,166.796,52.733,159.648
C04216=1019.319,52.226,-108.165,166.798,52.726,159.647
C04217=1019.325,52.475,-108.181,166.801,52.720,159.646
C04218=1019.330,52.724,-108.196,166.804,52.713,159.646
C04219=1019.335,52.974,-108.213,166.806,52.707,159.645
C04220=1019.341,53.224,-108.229,166.808,52.700,159.644
C04221=1019.347,53.473,-108.245,166.812,52.694,159.644
C04222=1019.352,53.722,-108.261,166.814,52.688,159.643
C04223=1019.358,53.972,-108.276,166.816,52.681,159.642
C04224=1019.364,54.221,-108.293,166.819,52.675,159.641
C04225=1019.369,54.470,-108.308,166.822,52.668,159.641
C04226=1019.375,54.720,-108.324,166.825,52.662,159.640
C04227=1019.381,54.970,-108.340,166.827,52.655,159.639
C04228=1019.386,55.218,-108.355,166.830,52.648,159.638
C04229=1019.392,55.468,-108.372,166.832,52.642,159.638
C04230=1019.397,55.718,-108.388,166.835,52.635,159.637
C04231=1019.403,55.967,-108.404,166.837,52.629,159.636
C04232=1019.408,56.217,-108.419,166.840,52.622,159.635
C04233=1019.414,56.466,-108.435,166.843,52.616,159.635
C04234=1019.420,56.715,-108.452,166.845,52.609,159.634
C04235=1019.425,56.964,-108.467,166.848,52.603,159.633
C04236=1019.431,57.214,-108.483,166.851,52.596,159.632
C04237=1019.437,57.463,-108.499,166.853,52.590,159.632
C04238=1019.442,57.713,-108.515,166.855,52.583,159.631
C04239=1019.448,57.962,-108.531,166.859,52.577,159.630
C04240=1019.453,58.212,-108.546,166.861,52.570,159.629
C04241=1019.459,58.461,-108.563,166.863,52.563,159.628
C04242=1019.465,58.744,-108.582,166.866,52.556,159.628
C04243=1019.472,59.027,-108.599,166.869,52.548,159.627
C04244=1019.478,59.311,-108.618,166.872,52.541,159.626
C04245=1019.484,59.592,-108.636,166.875,52.533,159.625
C04246=1019.490,59.842,-108.652,166.879,52.527,159.624
C04247=1019.496,60.092,-108.667,166.881,52.520,159.624
C04248=1019.502,60.341,-108.684,166.883,52.514,159.623
C04249=1019.507,60.591,-108.700,166.887,52.507,159.622
C04250=1019.512,60.840,-108.716,166.889,52.500,159.621
C04251=1019.518,61.089,-108.732,166.891,52.494,159.621
C04252=1019.524,61.339,-108.748,166.894,52.487,159.620
C04253=1019.530,61.588,-108.764,166.897,52.480,159.619
C04254=1019.536,61.838,-108.780,166.899,52.474,159.618
C04255=1019.541,62.087,-108.796,166.902,52.467,159.618
C04256=1019.547,62.336,-108.812,166.904,52.461,159.617
C04257=1019.553,62.585,-108.828,166.907,52.455,159.616
C04258=1019.558,62.836,-108.844,166.910,52.448,159.615
C04259=1019.564,63.085,-108.861,166.913,52.442,159.615
C04260=1019.570,63.334,-108.877,166.915,52.435,159.614
C04261=1019.575,63.584,-108.894,166.918,52.429,159.613
C04262=1019.580,63.833,-108.910,166.921,52.422,159.612
C04263=1019.586,64.082,-108.927,166.923,52.416,159.612
C04264=1019.591,64.332,-108.943,166.925,52.409,159.611
C04265=1019.597,64.581,-108.959,166.928,52.402,159.610
C04266=1019.603,64.831,-108.976,166.931,52.396,159.609
C04267=1019.609,65.080,-108.992,166.933,52.389,159.608
C04268=1019.614,65.330,-109.009,166.936,52.383,159.608
C04269=1019.619,65.578,-109.025,166.938,52.376,159.607
C04270=1019.624,65.828,-109.042,166.942,52.370,159.606
C04271=1019.630,66.077,-109.058,166.944,52.363,159.606
C04272=1019.636,66.327,-109.074,166.947,52.357,159.605
C04273=1019.641,66.576,-109.091,166.949,52.351,159.604
C04274=1019.647,66.826,-109.107,166.952,52.344,159.603
C04275=1019.653,67.075,-109.124,166.955,52.337,159.603
C04276=1019.658,67.324,-109.140,166.957,52.331,159.602
C04277=1019.663,67.574,-109.157,166.959,52.325,159.601
C04278=1019.669,67.823,-109.173,166.963,52.318,159.601
C04279=1019.674,68.073,-109.190,166.965,52.312,159.600
C04280=1019.680,68.322,-109.206,166.967,52.305,159.599
C04281=1019.686,68.572,-109.223,166.970,52.299,159.598
C04282=1019.691,68.821,-109.239,166.973,52.292,159.597
C04283=1019.697,69.071,-109.256,166.976,52.286,159.597
C04284=1019.702,69.320,-109.273,166.978,52.279,159.596
C04285=1019.708,69.570,-109.289,166.980,52.273,159.595
C04286=1019.713,69.818,-109.307,166.983,52.266,159.594
C04287=1019.718,70.068,-109.323,166.986,52.260,159.594
C04288=1019.724,70.317,-109.340,166.988,52.253,159.593
C04289=1019.729,70.567,-109.357,166.991,52.247,159.592
C04290=1019.735,70.816,-109.373,166.993,52.241,159.591
C04291=1019.740,71.066,-109.390,166.997,52.234,159.591
C04292=1019.746,71.315,-109.407,166.999,52.228,159.590
C04293=1019.752,71.564,-109.424,167.002,52.222,159.589
C04294=1019.757,71.814,-109.440,167.004,52.215,159.588
C04295=1019.762,72.063,-109.457,167.007,52.209,159.588
C04296=1019.768,72.313,-109.473,167.010,52.202,159.587
C04297=1019.774,72.562,-109.491,167.012,52.196,159.586
C04298=1019.779,72.811,-109.508,167.014,52.189,159.585
C04299=1019.785,73.061,-109.524,167.018,52.182,159.585
C04300=1019.790,73.311,-109.541,167.020,52.176,159.584
C04301=1019.796,73.560,-109.559,167.022,52.170,159.583
C04302=1019.802,73.809,-109.575,167.025,52.164,159.582
C04303=1019.806,74.058,-109.591,167.028,52.156,159.582
C04304=1019.812,74.307,-109.608,167.031,52.150,159.581
C04305=1019.818,74.556,-109.625,167.033,52.144,159.580
C04306=1019.824,74.840,-109.644,167.036,52.136,159.579
C04307=1019.831,75.123,-109.663,167.039,52.129,159.578
C04308=1019.837,75.405,-109.682,167.042,52.121,159.577
C04309=1019.843,75.688,-109.701,167.045,52.114,159.577
C04310=1019.849,75.937,-109.719,167.047,52.108,159.576
C04311=1019.854,76.187,-109.736,167.051,52.101,159.575
C04312=1019.860,76.436,-109.752,167.053,52.095,159.574
C04313=1019.865,76.685,-109.770,167.056,52.089,159.574
C04314=1019.870,76.935,-109.786,167.059,52.082,159.573
C04315=1019.876,77.184,-109.804,167.061,52.075,159.572
C04316=1019.881,77.434,-109.821,167.064,52.069,159.571
C04317=1019.886,77.683,-109.838,167.066,52.062,159.571
C04318=1019.892,77.932,-109.855,167.069,52.056,159.570
C04319=1019.898,78.182,-109.872,167.072,52.049,159.569
C04320=1019.903,78.431,-109.889,167.075,52.043,159.568
C04321=1019.909,78.681,-109.906,167.077,52.037,159.568
C04322=1019.914,78.930,-109.924,167.080,52.031,159.567
C04323=1019.919,79.179,-109.940,167.083,52.024,159.566
C04324=1019.925,79.428,-109.958,167.085,52.018,159.565
C04325=1019.930,79.678,-109.975,167.088,52.011,159.565
C04326=1019.936,79.927,-109.992,167.090,52.005,159.564
C04327=1019.941,80.176,-110.010,167.093,51.998,159.563
C04328=1019.946,80.426,-110.027,167.096,51.992,159.563
C04329=1019.952,80.675,-110.044,167.098,51.985,159.562
C04330=1019.957,80.924,-110.061,167.101,51.979,159.561
C04331=1019.963,81.173,-110.079,167.103,51.973,159.560
C04332=1019.968,81.424,-110.096,167.107,51.966,159.559
C04333=1019.974,81.673,-110.114,167.109,51.960,159.559
C04334=1019.979,81.922,-110.130,167.111,51.953,159.558
C04335=1019.985,82.172,-110.148,167.114,51.947,159.557
C04336=1019.990,82.421,-110.166,167.117,51.940,159.556
C04337=1019.995,82.670,-110.182,167.120,51.933,159.556
C04338=1020.002,82.919,-110.199,167.122,51.927,159.555
C04339=1020.007,83.169,-110.216,167.125,51.920,159.554
C04340=1020.012,83.418,-110.234,167.128,51.914,159.553
C04341=1020.018,83.667,-110.251,167.130,51.908,159.553
C04342=1020.024,83.917,-110.269,167.133,51.901,159.552
C04343=1020.029,84.166,-110.286,167.136,51.895,159.551
C04344=1020.035,84.415,-110.304,167.138,51.888,159.550
C04345=1020.040,84.665,-110.321,167.141,51.882,159.549
C04346=1020.045,84.914,-110.338,167.144,51.875,159.549
C04347=1020.051,85.163,-110.356,167.147,51.869,159.548
C04348=1020.056,85.413,-110.373,167.149,51.862,159.547
C04349=1020.062,85.662,-110.390,167.152,51.856,159.546
C04350=1020.068,85.911,-110.408,167.155,51.849,159.546
C04351=1020.073,86.161,-110.425,167.157,51.842,159.545
C04352=1020.079,86.410,-110.442,167.160,51.836,159.544
C04353=1020.084,86.659,-110.460,167.163,51.829,159.543
C04354=1020.089,86.909,-110.477,167.165,51.823,159.543
C04355=1020.095,87.158,-110.494,167.168,51.817,159.542
C04356=1020.101,87.407,-110.512,167.171,51.810,159.541
C04357=1020.106,87.657,-110.529,167.173,51.803,159.540
C04358=1020.112,87.906,-110.547,167.176,51.797,159.540
C04359=1020.117,88.155,-110.564,167.179,51.790,159.539
C04360=1020.123,88.404,-110.582,167.182,51.784,159.538
C04361=1020.128,88.654,-110.599,167.184,51.777,159.537
C04362=1020.134,88.904,-110.617,167.188,51.771,159.537
C04363=1020.140,89.153,-110.634,167.190,51.764,159.536
C04364=1020.145,89.402,-110.652,167.192,51.757,159.535
C04365=1020.151,89.651,-110.669,167.195,51.751,159.534
C04366=1020.156,89.901,-110.687,167.198,51.744,159.533
C04367=1020.161,90.151,-110.705,167.201,51.739,159.533
C04368=1020.167,90.400,-110.722,167.203,51.732,159.532
C04369=1020.172,90.649,-110.740,167.206,51.726,159.531
C04370=1020.178,90.931,-110.760,167.209,51.718,159.530
C04371=1020.184,91.214,-110.781,167.212,51.711,159.529
C04372=1020.190,91.497,-110.801,167.215,51.704,159.528
C04373=1020.197,91.780,-110.821,167.218,51.697,159.528
C04374=1020.202,92.030,-110.839,167.221,51.690,159.527
C04375=1020.207,92.279,-110.856,167.224,51.684,159.526
C04376=1020.213,92.528,-110.874,167.226,51.677,159.525
C04377=1020.219,92.778,-110.892,167.228,51.671,159.525
C04378=1020.224,93.027,-110.910,167.232,51.664,159.524
C04379=1020.229,93.276,-110.927,167.234,51.658,159.523
C04380=1020.235,93.525,-110.945,167.237,51.652,159.522
C04381=1020.241,93.775,-110.963,167.240,51.645,159.522
C04382=1020.246,94.024,-110.981,167.243,51.638,159.521
C04383=1020.251,94.273,-110.999,167.245,51.632,159.520
C04384=1020.257,94.522,-111.016,167.248,51.626,159.519
C04385=1020.262,94.772,-111.035,167.251,51.619,159.519
C04386=1020.268,95.021,-111.052,167.254,51.613,159.518
C04387=1020.273,95.270,-111.070,167.256,51.606,159.517
C04388=1020.279,95.519,-111.087,167.259,51.599,159.516
C04389=1020.284,95.769,-111.106,167.262,51.593,159.516
C04390=1020.290,96.018,-111.124,167.264,51.587,159.515
C04391=1020.295,96.267,-111.142,167.268,51.580,159.514
C04392=1020.301,96.517,-111.160,167.270,51.574,159.513
C04393=1020.306,96.766,-111.178,167.273,51.567,159.512
C04394=1020.312,97.015,-111.196,167.276,51.560,159.512
C04395=1020.317,97.264,-111.213,167.278,51.554,159.511
C04396=1020.323,97.514,-111.232,167.281,51.548,159.510
C04397=1020.328,97.763,-111.249,167.284,51.541,159.509
C04398=1020.334,98.012,-111.267,167.286,51.534,159.508
C04399=1020.339,98.262,-111.285,167.289,51.528,159.508
C04400=1020.345,98.511,-111.303,167.292,51.521,159.507
C04401=1020.350,98.760,-111.320,167.295,51.515,159.506
C04402=1020.356,99.010,-111.340,167.297,51.508,159.505
C04403=1020.361,99.259,-111.357,167.301,51.502,159.505
C04404=1020.367,99.508,-111.375,167.303,51.495,159.504
C04405=1020.372,99.758,-111.393,167.306,51.489,159.503
C04406=1020.377,100.007,-111.411,167.309,51.482,159.502
C04407=1020.383,100.256,-111.430,167.311,51.476,159.502
C04408=1020.388,100.506,-111.448,167.314,51.470,159.501
C04409=1020.394,100.755,-111.466,167.316,51.463,159.500
C04410=1020.399,101.004,-111.485,167.320,51.457,159.500
C04411=1020.405,101.253,-111.503,167.322,51.450,159.499
C04412=1020.410,101.503,-111.521,167.325,51.444,159.498
C04413=1020.415,101.752,-111.540,167.329,51.438,159.497
C04414=1020.421,102.001,-111.558,167.331,51.431,159.496
C04415=1020.426,102.250,-111.576,167.334,51.425,159.496
C04416=1020.432,102.500,-111.594,167.337,51.418,159.495
C04417=1020.437,102.749,-111.613,167.339,51.412,159.494
C04418=1020.442,102.998,-111.631,167.342,51.406,159.493
C04419=1020.448,103.247,-111.649,167.344,51.399,159.493
C04420=1020.453,103.497,-111.668,167.348,51.392,159.492
C04421=1020.459,103.746,-111.686,167.350,51.386,159.491
C04422=1020.464,103.995,-111.704,167.353,51.380,159.490
C04423=1020.470,104.244,-111.722,167.356,51.373,159.490
C04424=1020.475,104.494,-111.740,167.359,51.367,159.489
C04425=1020.480,104.743,-111.759,167.361,51.360,159.488
C04426=1020.486,104.993,-111.777,167.365,51.354,159.487
C04427=1020.491,105.242,-111.796,167.367,51.347,159.487
C04428=1020.497,105.491,-111.814,167.369,51.341,159.486
C04429=1020.502,105.741,-111.832,167.373,51.335,159.485
C04430=1020.507,105.989,-111.851,167.375,51.328,159.484
C04431=1020.513,106.239,-111.869,167.378,51.321,159.483
C04432=1020.519,106.488,-111.888,167.381,51.315,159.483
C04433=1020.525,106.738,-111.906,167.384,51.309,159.482
C04434=1020.530,107.020,-111.927,167.387,51.301,159.481
C04435=1020.536,107.303,-111.948,167.390,51.294,159.480
C04436=1020.543,107.586,-111.969,167.393,51.287,159.479
C04437=1020.549,107.870,-111.989,167.397,51.279,159.478
C04438=1020.554,108.118,-112.008,167.400,51.273,159.478
C04439=1020.560,108.368,-112.026,167.402,51.266,159.477
C04440=1020.565,108.617,-112.045,167.405,51.259,159.476
C04441=1020.572,108.866,-112.063,167.408,51.253,159.475
C04442=1020.577,109.115,-112.082,167.411,51.247,159.475
C04443=1020.582,109.365,-112.100,167.414,51.240,159.474
C04444=1020.588,109.614,-112.119,167.416,51.233,159.473
C04445=1020.593,109.864,-112.137,167.420,51.227,159.472
C04446=1020.598,110.112,-112.156,167.422,51.221,159.472
C04447=1020.604,110.362,-112.175,167.425,51.214,159.471
C04448=1020.609,110.611,-112.193,167.428,51.208,159.470
C04449=1020.615,110.860,-112.212,167.431,51.201,159.469
C04450=1020.620,111.109,-112.231,167.433,51.195,159.468
C04451=1020.626,111.359,-112.250,167.437,51.188,159.468
C04452=1020.631,111.608,-112.268,167.439,51.182,159.467
C04453=1020.637,111.858,-112.286,167.442,51.175,159.466
C04454=1020.642,112.106,-112.305,167.445,51.169,159.466
C04455=1020.648,112.356,-112.325,167.448,51.163,159.465
C04456=1020.653,112.605,-112.343,167.450,51.156,159.464
C04457=1020.658,112.855,-112.362,167.454,51.150,159.463
C04458=1020.663,113.103,-112.381,167.456,51.143,159.462
C04459=1020.669,113.353,-112.400,167.459,51.137,159.462
C04460=1020.674,113.601,-112.419,167.462,51.131,159.461
C04461=1020.680,113.851,-112.438,167.465,51.125,159.460
C04462=1020.684,114.100,-112.456,167.467,51.118,159.459
C04463=1020.690,114.350,-112.476,167.471,51.112,159.459
C04464=1020.694,114.599,-112.495,167.474,51.105,159.458
C04465=1020.700,114.848,-112.514,167.476,51.100,159.457
C04466=1020.705,115.097,-112.533,167.479,51.093,159.456
C04467=1020.711,115.346,-112.552,167.482,51.087,159.456
C04468=1020.716,115.595,-112.571,167.485,51.080,159.455
C04469=1020.721,115.845,-112.590,167.488,51.074,159.454
C04470=1020.727,116.095,-112.609,167.491,51.068,159.454
C04471=1020.732,116.343,-112.628,167.493,51.061,159.453
C04472=1020.738,116.593,-112.647,167.496,51.055,159.452
C04473=1020.743,116.841,-112.666,167.500,51.048,159.451
C04474=1020.749,117.091,-112.685,167.502,51.042,159.451
C04475=1020.754,117.340,-112.704,167.505,51.036,159.450
C04476=1020.759,117.589,-112.723,167.508,51.029,159.449
C04477=1020.764,117.839,-112.743,167.511,51.023,159.448
C04478=1020.769,118.088,-112.762,167.513,51.017,159.447
C04479=1020.775,118.338,-112.781,167.517,51.011,159.447
C04480=1020.780,118.586,-112.800,167.519,51.004,159.446
C04481=1020.786,118.836,-112.819,167.523,50.997,159.445
C04482=1020.791,119.085,-112.838,167.525,50.991,159.445
C04483=1020.796,119.334,-112.857,167.528,50.985,159.444
C04484=1020.802,119.583,-112.876,167.532,50.979,159.443
C04485=1020.807,119.832,-112.895,167.534,50.972,159.442
C04486=1020.813,120.081,-112.914,167.536,50.966,159.441
C04487=1020.819,120.331,-112.934,167.540,50.959,159.441
C04488=1020.824,120.580,-112.952,167.543,50.953,159.440
C04489=1020.829,120.829,-112.972,167.546,50.946,159.439
C04490=1020.834,121.079,-112.991,167.549,50.940,159.439
C04491=1020.839,121.328,-113.010,167.551,50.934,159.438
C04492=1020.845,121.577,-113.030,167.555,50.927,159.437
C04493=1020.851,121.826,-113.049,167.557,50.921,159.436
C04494=1020.856,122.075,-113.068,167.561,50.914,159.436
C04495=1020.861,122.325,-113.087,167.564,50.908,159.435
C04496=1020.867,122.574,-113.106,167.566,50.902,159.434
C04497=1020.873,122.822,-113.126,167.569,50.895,159.433
C04498=1020.878,123.106,-113.147,167.573,50.888,159.432
C04499=1020.884,123.389,-113.169,167.576,50.881,159.432
C04500=1020.891,123.672,-113.191,167.579,50.874,159.431
C04501=1020.897,123.955,-113.213,167.583,50.866,159.430
C04502=1020.903,124.203,-113.232,167.586,50.859,159.429
C04503=1020.908,124.452,-113.252,167.588,50.853,159.428
C04504=1020.913,124.702,-113.271,167.592,50.847,159.428
C04505=1020.919,124.952,-113.291,167.594,50.840,159.427
C04506=1020.924,125.200,-113.309,167.598,50.833,159.426
C04507=1020.930,125.450,-113.329,167.600,50.827,159.425
C04508=1020.936,125.699,-113.348,167.604,50.821,159.425
C04509=1020.941,125.948,-113.367,167.606,50.814,159.424
C04510=1020.947,126.197,-113.387,167.610,50.808,159.423
C04511=1020.952,126.446,-113.406,167.612,50.801,159.422
C04512=1020.958,126.696,-113.425,167.616,50.795,159.421
C04513=1020.963,126.944,-113.444,167.619,50.789,159.421
C04514=1020.968,127.194,-113.464,167.622,50.782,159.420
C04515=1020.974,127.444,-113.483,167.625,50.775,159.419
C04516=1020.980,127.692,-113.503,167.628,50.769,159.418
C04517=1020.985,127.942,-113.522,167.631,50.763,159.418
C04518=1020.991,128.191,-113.541,167.634,50.756,159.417
C04519=1020.996,128.440,-113.561,167.637,50.750,159.416
C04520=1021.002,128.689,-113.580,167.640,50.743,159.415
C04521=1021.008,128.938,-113.600,167.643,50.737,159.415
C04522=1021.013,129.187,-113.619,167.646,50.730,159.414
C04523=1021.018,129.437,-113.638,167.649,50.724,159.413
C04524=1021.024,129.686,-113.658,167.652,50.717,159.412
C04525=1021.030,129.935,-113.678,167.655,50.711,159.412
C04526=1021.035,130.184,-113.697,167.657,50.704,159.411
C04527=1021.040,130.433,-113.716,167.661,50.698,159.410
C04528=1021.046,130.682,-113.736,167.664,50.692,159.409
C04529=1021.051,130.932,-113.756,167.667,50.685,159.409
C04530=1021.057,131.181,-113.776,167.670,50.679,159.408
C04531=1021.062,131.430,-113.795,167.673,50.672,159.407
C04532=1021.067,131.679,-113.816,167.676,50.667,159.406
C04533=1021.073,131.928,-113.835,167.680,50.660,159.406
C04534=1021.078,132.177,-113.855,167.682,50.654,159.405
C04535=1021.084,132.427,-113.875,167.685,50.648,159.404
C04536=1021.089,132.676,-113.894,167.688,50.641,159.403
C04537=1021.094,132.924,-113.914,167.691,50.635,159.403
C04538=1021.099,133.174,-113.934,167.695,50.628,159.402
C04539=1021.105,133.423,-113.954,167.697,50.622,159.401
C04540=1021.110,133.673,-113.974,167.701,50.616,159.401
C04541=1021.116,133.922,-113.994,167.703,50.609,159.400
C04542=1021.121,134.171,-114.013,167.707,50.603,159.399
C04543=1021.127,134.420,-114.033,167.710,50.596,159.398
C04544=1021.132,134.669,-114.052,167.713,50.590,159.398
C04545=1021.137,134.918,-114.073,167.716,50.584,159.397
C04546=1021.143,135.167,-114.093,167.719,50.577,159.396
C04547=1021.148,135.417,-114.113,167.722,50.571,159.395
C04548=1021.154,135.665,-114.133,167.726,50.565,159.395
C04549=1021.159,135.915,-114.152,167.728,50.558,159.394
C04550=1021.165,136.164,-114.172,167.732,50.552,159.393
C04551=1021.170,136.414,-114.192,167.734,50.545,159.392
C04552=1021.175,136.662,-114.212,167.737,50.540,159.392
C04553=1021.181,136.911,-114.232,167.741,50.533,159.391
C04554=1021.186,137.160,-114.252,167.743,50.527,159.390
C04555=1021.192,137.409,-114.272,167.747,50.520,159.389
C04556=1021.197,137.659,-114.293,167.749,50.514,159.389
C04557=1021.202,137.908,-114.312,167.753,50.508,159.388
C04558=1021.208,138.157,-114.333,167.756,50.501,159.387
C04559=1021.214,138.406,-114.353,167.759,50.495,159.387
C04560=1021.219,138.656,-114.372,167.762,50.489,159.386
C04561=1021.224,138.905,-114.393,167.766,50.483,159.385
C04562=1021.230,139.187,-114.416,167.769,50.475,159.384
C04563=1021.236,139.470,-114.439,167.772,50.468,159.383
C04564=1021.242,139.753,-114.461,167.776,50.461,159.383
C04565=1021.248,140.036,-114.484,167.780,50.454,159.382
C04566=1021.254,140.285,-114.504,167.782,50.447,159.381
C04567=1021.259,140.534,-114.525,167.786,50.441,159.380
C04568=1021.264,140.783,-114.546,167.789,50.435,159.380
C04569=1021.269,141.033,-114.565,167.793,50.429,159.379
C04570=1021.275,141.282,-114.585,167.795,50.422,159.378
C04571=1021.280,141.531,-114.606,167.799,50.416,159.378
C04572=1021.286,141.780,-114.626,167.801,50.410,159.377
C04573=1021.291,142.029,-114.647,167.805,50.404,159.376
C04574=1021.297,142.278,-114.667,167.808,50.397,159.375
C04575=1021.302,142.528,-114.687,167.812,50.391,159.375
C04576=1021.307,142.777,-114.707,167.814,50.385,159.374
C04577=1021.313,143.026,-114.727,167.818,50.379,159.373
C04578=1021.318,143.275,-114.748,167.820,50.372,159.372
C04579=1021.324,143.524,-114.768,167.824,50.365,159.372
C04580=1021.329,143.773,-114.789,167.827,50.360,159.371
C04581=1021.335,144.022,-114.809,167.830,50.353,159.370
C04582=1021.340,144.271,-114.829,167.834,50.347,159.370
C04583=1021.345,144.520,-114.850,167.837,50.340,159.369
C04584=1021.351,144.769,-114.871,167.840,50.334,159.368
C04585=1021.356,145.019,-114.890,167.843,50.328,159.367
C04586=1021.362,145.268,-114.910,167.846,50.321,159.367
C04587=1021.367,145.517,-114.931,167.849,50.315,159.366
C04588=1021.372,145.766,-114.951,167.853,50.309,159.365
C04589=1021.378,146.015,-114.971,167.856,50.303,159.364
C04590=1021.383,146.264,-114.992,167.859,50.296,159.364
C04591=1021.389,146.513,-115.013,167.863,50.290,159.363
C04592=1021.394,146.762,-115.033,167.865,50.284,159.362
C04593=1021.399,147.011,-115.054,167.869,50.278,159.362
C04594=1021.405,147.260,-115.075,167.872,50.271,159.361
C04595=1021.411,147.510,-115.096,167.876,50.265,159.360
C04596=1021.416,147.759,-115.116,167.878,50.259,159.359
C04597=1021.421,148.008,-115.137,167.882,50.253,159.359
C04598=1021.426,148.257,-115.157,167.885,50.247,159.358
C04599=1021.432,148.506,-115.178,167.888,50.240,159.357
C04600=1021.437,148.755,-115.199,167.891,50.234,159.357
C04601=1021.442,149.004,-115.219,167.895,50.228,159.356
C04602=1021.448,149.253,-115.240,167.898,50.222,159.355
C04603=1021.453,149.502,-115.261,167.901,50.215,159.355
C04604=1021.458,149.751,-115.282,167.905,50.209,159.354
C04605=1021.463,150.000,-115.302,167.908,50.203,159.353
C04606=1021.469,150.250,-115.323,167.911,50.197,159.353
C04607=1021.475,150.498,-115.344,167.914,50.190,159.352
C04608=1021.480,150.748,-115.365,167.918,50.184,159.351
C04609=1021.485,150.997,-115.385,167.920,50.178,159.350
C04610=1021.491,151.246,-115.406,167.924,50.172,159.350
C04611=1021.496,151.495,-115.426,167.928,50.165,159.349
C04612=1021.501,151.743,-115.448,167.931,50.159,159.348
C04613=1021.507,151.993,-115.468,167.935,50.153,159.348
C04614=1021.513,152.242,-115.489,167.937,50.147,159.347
C04615=1021.518,152.492,-115.510,167.941,50.141,159.346
C04616=1021.523,152.740,-115.531,167.944,50.134,159.345
C04617=1021.529,152.989,-115.552,167.947,50.128,159.345
C04618=1021.534,153.238,-115.572,167.951,50.122,159.344
C04619=1021.539,153.487,-115.593,167.954,50.116,159.343
C04620=1021.545,153.737,-115.614,167.957,50.109,159.343
C04621=1021.551,153.986,-115.635,167.960,50.104,159.342
C04622=1021.555,154.235,-115.657,167.964,50.097,159.341
C04623=1021.561,154.484,-115.677,167.968,50.091,159.341
C04624=1021.566,154.732,-115.699,167.970,50.085,159.340
C04625=1021.572,154.982,-115.720,167.974,50.078,159.339
C04626=1021.578,155.264,-115.743,167.977,50.072,159.338
C04627=1021.584,155.547,-115.767,167.982,50.065,159.338
C04628=1021.590,155.829,-115.791,167.985,50.057,159.337
C04629=1021.596,156.113,-115.815,167.989,50.050,159.336
C04630=1021.601,156.361,-115.836,167.993,50.044,159.335
C04631=1021.607,156.610,-115.857,167.996,50.038,159.335
C04632=1021.613,156.860,-115.878,167.999,50.032,159.334
C04633=1021.617,157.109,-115.899,168.003,50.026,159.333
C04634=1021.623,157.357,-115.921,168.006,50.020,159.332
C04635=1021.628,157.607,-115.941,168.009,50.014,159.332
C04636=1021.634,157.855,-115.962,168.013,50.007,159.331
C04637=1021.640,158.105,-115.983,168.016,50.001,159.330
C04638=1021.645,158.353,-116.005,168.019,49.994,159.330
C04639=1021.650,158.603,-116.026,168.023,49.988,159.329
C04640=1021.656,158.852,-116.047,168.026,49.983,159.328
C04641=1021.661,159.101,-116.068,168.030,49.976,159.328
C04642=1021.666,159.350,-116.090,168.033,49.970,159.327
C04643=1021.672,159.599,-116.111,168.037,49.964,159.326
C04644=1021.677,159.848,-116.133,168.039,49.959,159.326
C04645=1021.681,160.097,-116.154,168.043,49.952,159.325
C04646=1021.687,160.346,-116.176,168.047,49.946,159.324
C04647=1021.692,160.595,-116.198,168.050,49.940,159.324
C04648=1021.697,160.844,-116.220,168.054,49.934,159.323
C04649=1021.703,161.093,-116.241,168.057,49.929,159.322
C04650=1021.707,161.342,-116.262,168.061,49.923,159.322
C04651=1021.712,161.591,-116.284,168.063,49.916,159.321
C04652=1021.718,161.840,-116.306,168.067,49.910,159.320
C04653=1021.723,162.089,-116.328,168.071,49.904,159.320
C04654=1021.729,162.338,-116.349,168.074,49.899,159.319
C04655=1021.734,162.586,-116.371,168.078,49.893,159.319
C04656=1021.739,162.837,-116.392,168.080,49.886,159.318
C04657=1021.744,163.085,-116.414,168.084,49.880,159.317
C04658=1021.749,163.334,-116.435,168.088,49.874,159.317
C04659=1021.755,163.583,-116.458,168.091,49.868,159.316
C04660=1021.760,163.832,-116.479,168.095,49.862,159.315
C04661=1021.765,164.081,-116.501,168.098,49.856,159.314
C04662=1021.770,164.330,-116.523,168.102,49.850,159.314
C04663=1021.776,164.579,-116.544,168.105,49.844,159.313
C04664=1021.780,164.828,-116.565,168.108,49.838,159.313
C04665=1021.787,165.077,-116.587,168.112,49.832,159.312
C04666=1021.791,165.326,-116.609,168.116,49.826,159.311
C04667=1021.796,165.575,-116.631,168.119,49.820,159.311
C04668=1021.802,165.824,-116.652,168.123,49.814,159.310
C04669=1021.807,166.073,-116.674,168.126,49.808,159.309
C04670=1021.813,166.323,-116.697,168.129,49.802,159.309
C04671=1021.818,166.571,-116.718,168.133,49.796,159.308
C04672=1021.823,166.820,-116.740,168.136,49.790,159.307
C04673=1021.828,167.069,-116.762,168.140,49.784,159.307
C04674=1021.834,167.318,-116.783,168.144,49.778,159.306
C04675=1021.839,167.567,-116.805,168.146,49.772,159.305
C04676=1021.844,167.816,-116.827,168.150,49.766,159.305
C04677=1021.850,168.065,-116.849,168.154,49.760,159.304
C04678=1021.855,168.314,-116.871,168.157,49.754,159.304
C04679=1021.860,168.563,-116.893,168.161,49.748,159.303
C04680=1021.866,168.812,-116.914,168.165,49.742,159.302
C04681=1021.871,169.061,-116.936,168.169,49.736,159.302
C04682=1021.876,169.311,-116.958,168.172,49.730,159.301
C04683=1021.882,169.559,-116.980,168.176,49.724,159.300
C04684=1021.887,169.807,-117.002,168.179,49.717,159.300
C04685=1021.893,170.057,-117.024,168.182,49.712,159.299
C04686=1021.898,170.305,-117.046,168.186,49.706,159.298
C04687=1021.904,170.555,-117.068,168.190,49.700,159.298
C04688=1021.908,170.804,-117.090,168.194,49.693,159.297
C04689=1021.915,171.053,-117.111,168.197,49.687,159.296
C04690=1021.921,171.335,-117.137,168.201,49.680,159.296
C04691=1021.926,171.617,-117.161,168.205,49.674,159.295
C04692=1021.933,171.899,-117.186,168.209,49.667,159.294
C04693=1021.939,172.182,-117.211,168.213,49.660,159.293
C04694=1021.945,172.430,-117.233,168.217,49.654,159.293
C04695=1021.950,172.680,-117.255,168.221,49.648,159.292
C04696=1021.955,172.929,-117.277,168.224,49.642,159.291
C04697=1021.961,173.178,-117.299,168.228,49.636,159.291
C04698=1021.966,173.427,-117.321,168.231,49.630,159.290
C04699=1021.972,173.675,-117.344,168.235,49.624,159.290
C04700=1021.978,173.925,-117.365,168.239,49.617,159.289
C04701=1021.983,174.173,-117.387,168.243,49.611,159.288
C04702=1021.988,174.423,-117.409,168.246,49.606,159.288
C04703=1021.993,174.671,-117.432,168.250,49.600,159.287
C04704=1021.999,174.920,-117.454,168.253,49.593,159.286
C04705=1022.005,175.170,-117.476,168.257,49.587,159.286
C04706=1022.010,175.419,-117.498,168.261,49.581,159.285
C04707=1022.016,175.667,-117.520,168.265,49.575,159.284
C04708=1022.021,175.916,-117.542,168.268,49.570,159.284
C04709=1022.026,176.166,-117.564,168.272,49.563,159.283
C04710=1022.033,176.414,-117.586,168.276,49.557,159.282
C04711=1022.038,176.663,-117.608,168.280,49.551,159.282
C04712=1022.043,176.913,-117.631,168.284,49.545,159.281
C04713=1022.049,177.160,-117.653,168.287,49.539,159.280
C04714=1022.054,177.410,-117.675,168.290,49.533,159.280
C04715=1022.060,177.660,-117.697,168.294,49.527,159.279
C04716=1022.066,177.907,-117.719,168.298,49.521,159.279
C04717=1022.071,178.157,-117.741,168.302,49.515,159.278
C04718=1022.076,178.406,-117.763,168.306,49.509,159.277
C04719=1022.082,178.654,-117.785,168.310,49.503,159.277
C04720=1022.088,178.904,-117.808,168.314,49.497,159.276
C04721=1022.093,179.153,-117.831,168.318,49.491,159.275
C04722=1022.099,179.402,-117.853,168.321,49.485,159.275
C04723=1022.105,179.650,-117.875,168.324,49.479,159.274
C04724=1022.110,179.900,-117.897,168.328,49.473,159.273
C04725=1022.116,180.149,-117.919,168.332,49.467,159.273
C04726=1022.121,180.397,-117.941,168.336,49.461,159.272
C04727=1022.127,180.647,-117.963,168.340,49.454,159.272
C04728=1022.133,180.895,-117.986,168.344,49.448,159.271
C04729=1022.139,181.145,-118.008,168.348,49.442,159.270
C04730=1022.144,181.393,-118.031,168.352,49.436,159.270
C04731=1022.149,181.642,-118.053,168.356,49.430,159.269
C04732=1022.155,181.891,-118.076,168.359,49.424,159.268
C04733=1022.161,182.140,-118.097,168.362,49.418,159.268
C04734=1022.166,182.389,-118.120,168.366,49.412,159.267
C04735=1022.171,182.638,-118.144,168.370,49.406,159.267
C04736=1022.177,182.887,-118.166,168.374,49.400,159.266
C04737=1022.183,183.136,-118.189,168.378,49.395,159.265
C04738=1022.187,183.385,-118.212,168.382,49.390,159.265
C04739=1022.193,183.634,-118.235,168.386,49.384,159.264
C04740=1022.198,183.883,-118.258,168.389,49.378,159.264
C04741=1022.203,184.132,-118.281,168.393,49.372,159.263
C04742=1022.208,184.381,-118.303,168.397,49.366,159.263
C04743=1022.214,184.630,-118.326,168.400,49.360,159.262
C04744=1022.219,184.879,-118.350,168.404,49.354,159.261
C04745=1022.225,185.128,-118.373,168.408,49.348,159.261
C04746=1022.230,185.376,-118.395,168.413,49.343,159.260
C04747=1022.235,185.625,-118.419,168.417,49.337,159.260
C04748=1022.240,185.874,-118.442,168.421,49.331,159.259
C04749=1022.246,186.123,-118.465,168.424,49.326,159.258
C04750=1022.251,186.371,-118.488,168.428,49.320,159.258
C04751=1022.256,186.620,-118.511,168.432,49.314,159.257
C04752=1022.262,186.869,-118.534,168.436,49.308,159.257
C04753=1022.267,187.118,-118.557,168.440,49.302,159.256
C04754=1022.273,187.401,-118.583,168.445,49.296,159.256
C04755=1022.279,187.682,-118.609,168.448,49.289,159.255
C04756=1022.285,187.964,-118.635,168.453,49.283,159.254
C04757=1022.291,188.245,-118.662,168.457,49.277,159.253
C04758=1022.297,188.496,-118.684,168.461,49.271,159.253
C04759=1022.302,188.745,-118.707,168.465,49.265,159.252
C04760=1022.308,188.995,-118.731,168.469,49.259,159.252
C04761=1022.313,189.246,-118.754,168.473,49.253,159.251
C04762=1022.319,189.494,-118.778,168.477,49.247,159.250
C04763=1022.324,189.742,-118.800,168.481,49.242,159.250
C04764=1022.329,189.992,-118.824,168.485,49.236,159.250
C04765=1022.335,190.240,-118.847,168.489,49.230,159.249
C04766=1022.341,190.489,-118.870,168.493,49.224,159.248
C04767=1022.346,190.739,-118.893,168.497,49.218,159.248
C04768=1022.351,190.987,-118.916,168.501,49.212,159.247
C04769=1022.357,191.236,-118.939,168.505,49.207,159.247
C04770=1022.362,191.486,-118.963,168.510,49.201,159.246
C04771=1022.368,191.734,-118.987,168.513,49.196,159.245
C04772=1022.374,191.983,-119.009,168.517,49.190,159.245
C04773=1022.378,192.231,-119.033,168.521,49.184,159.244
C04774=1022.384,192.480,-119.056,168.525,49.178,159.244
C04775=1022.389,192.729,-119.079,168.529,49.172,159.243
C04776=1022.395,192.978,-119.103,168.533,49.167,159.243
C04777=1022.401,193.226,-119.126,168.537,49.161,159.242
C04778=1022.406,193.476,-119.149,168.541,49.155,159.241
C04779=1022.411,193.725,-119.172,168.545,49.149,159.241
C04780=1022.417,193.974,-119.195,168.549,49.144,159.240
C04781=1022.422,194.222,-119.219,168.553,49.138,159.240
C04782=1022.428,194.471,-119.242,168.558,49.133,159.239
C04783=1022.434,194.720,-119.265,168.562,49.127,159.239
C04784=1022.439,194.968,-119.290,168.566,49.121,159.238
C04785=1022.445,195.217,-119.313,168.570,49.115,159.237
C04786=1022.450,195.467,-119.336,168.574,49.109,159.237
C04787=1022.456,195.715,-119.359,168.578,49.103,159.236
C04788=1022.462,195.964,-119.383,168.582,49.098,159.236
C04789=1022.467,196.213,-119.406,168.586,49.092,159.235
C04790=1022.473,196.463,-119.430,168.590,49.086,159.235
C04791=1022.479,196.711,-119.453,168.595,49.080,159.234
C04792=1022.484,196.960,-119.477,168.599,49.074,159.234
C04793=1022.490,197.208,-119.500,168.603,49.069,159.233
C04794=1022.496,197.457,-119.523,168.607,49.063,159.233
C04795=1022.501,197.706,-119.547,168.611,49.057,159.232
C04796=1022.507,197.955,-119.571,168.615,49.051,159.231
C04797=1022.512,198.204,-119.594,168.619,49.046,159.231
C04798=1022.518,198.452,-119.618,168.624,49.040,159.230
C04799=1022.524,198.701,-119.641,168.628,49.035,159.230
C04800=1022.529,198.950,-119.665,168.632,49.029,159.229
C04801=1022.535,199.199,-119.688,168.636,49.023,159.229
C04802=1022.541,199.448,-119.712,168.640,49.018,159.228
C04803=1022.546,199.697,-119.735,168.644,49.012,159.228
C04804=1022.552,199.945,-119.760,168.649,49.006,159.227
C04805=1022.557,200.194,-119.783,168.653,49.000,159.226
C04806=1022.563,200.443,-119.807,168.658,48.995,159.226
C04807=1022.568,200.691,-119.831,168.662,48.989,159.225
C04808=1022.573,200.941,-119.855,168.666,48.984,159.225
C04809=1022.579,201.190,-119.879,168.670,48.978,159.224
C04810=1022.585,201.438,-119.903,168.675,48.973,159.224
C04811=1022.590,201.687,-119.927,168.679,48.967,159.223
C04812=1022.595,201.936,-119.951,168.683,48.961,159.223
C04813=1022.601,202.184,-119.974,168.687,48.956,159.222
C04814=1022.607,202.434,-119.999,168.691,48.950,159.222
C04815=1022.612,202.683,-120.023,168.695,48.945,159.221
C04816=1022.617,202.931,-120.047,168.699,48.939,159.221
C04817=1022.623,203.180,-120.071,168.703,48.933,159.220
C04818=1022.651,204.420,-120.192,169.131,49.027,159.304
C04819=1022.657,204.630,-120.213,169.135,49.023,159.304
C04820=1022.662,204.842,-120.235,169.137,49.019,159.304
C04821=1022.668,205.053,-120.256,169.139,49.014,159.303
C04822=1022.673,205.264,-120.278,169.142,49.010,159.303
C04823=1022.679,205.475,-120.300,169.145,49.007,159.302
C04824=1022.684,205.686,-120.322,169.148,49.002,159.302
C04825=1022.689,205.898,-120.343,169.151,48.998,159.301
C04826=1022.696,206.146,-120.370,169.155,48.994,159.301
C04827=1022.702,206.395,-120.395,169.158,48.989,159.301
C04828=1022.709,206.644,-120.421,169.160,48.985,159.300
C04829=1022.715,206.892,-120.447,169.164,48.981,159.300
C04830=1022.721,207.140,-120.472,169.167,48.976,159.299
C04831=1022.728,207.389,-120.497,169.171,48.971,159.298
C04832=1022.735,207.638,-120.524,169.174,48.967,159.298
C04833=1022.741,207.887,-120.549,169.178,48.962,159.298
C04834=1022.747,208.135,-120.575,169.181,48.957,159.297
C04835=1022.753,208.384,-120.601,169.185,48.953,159.297
C04836=1022.759,208.632,-120.626,169.188,48.948,159.296
C04837=1022.766,208.881,-120.653,169.192,48.944,159.296
C04838=1022.772,209.130,-120.678,169.194,48.939,159.295
C04839=1022.779,209.378,-120.704,169.197,48.935,159.295
C04840=1022.785,209.626,-120.730,169.201,48.930,159.294
C04841=1022.792,209.875,-120.756,169.204,48.925,159.294
C04842=1022.798,210.124,-120.782,169.208,48.921,159.293
C04843=1022.804,210.372,-120.808,169.211,48.916,159.293
C04844=1022.810,210.621,-120.833,169.215,48.912,159.293
C04845=1022.816,210.869,-120.860,169.218,48.907,159.292
C04846=1022.823,211.118,-120.886,169.221,48.904,159.292
C04847=1022.829,211.367,-120.912,169.224,48.899,159.291
C04848=1022.835,211.615,-120.938,169.228,48.895,159.291
C04849=1022.841,211.864,-120.964,169.232,48.890,159.290
C04850=1022.849,212.112,-120.990,169.235,48.886,159.290
C04851=1022.854,212.361,-121.017,169.239,48.881,159.290
C04852=1022.861,212.609,-121.042,169.242,48.877,159.289
C04853=1022.867,212.857,-121.068,169.245,48.873,159.289
C04854=1022.873,213.106,-121.095,169.249,48.869,159.288
C04855=1022.880,213.355,-121.120,169.252,48.864,159.288
C04856=1022.886,213.603,-121.147,169.256,48.859,159.287
C04857=1022.892,213.852,-121.174,169.259,48.855,159.287
C04858=1022.899,214.101,-121.199,169.263,48.850,159.286
C04859=1022.905,214.349,-121.225,169.266,48.846,159.286
C04860=1022.911,214.597,-121.252,169.269,48.842,159.286
C04861=1022.918,214.847,-121.277,169.272,48.838,159.285
C04862=1022.924,215.095,-121.303,169.276,48.833,159.285
C04863=1022.930,215.343,-121.330,169.279,48.829,159.284
C04864=1022.937,215.592,-121.356,169.283,48.824,159.284
C04865=1022.943,215.841,-121.382,169.287,48.820,159.284
C04866=1022.950,216.090,-121.409,169.290,48.815,159.283
C04867=1022.956,216.338,-121.435,169.293,48.812,159.283
C04868=1022.962,216.586,-121.461,169.296,48.807,159.282
C04869=1022.969,216.835,-121.488,169.300,48.803,159.282
C04870=1022.975,217.083,-121.513,169.303,48.798,159.281
C04871=1022.981,217.332,-121.540,169.307,48.794,159.281
C04872=1022.988,217.581,-121.566,169.311,48.790,159.281
C04873=1022.995,217.829,-121.592,169.314,48.785,159.280
C04874=1023.001,218.078,-121.619,169.317,48.781,159.280
C04875=1023.008,218.326,-121.645,169.321,48.777,159.279
C04876=1023.014,218.574,-121.671,169.324,48.773,159.279
C04877=1023.020,218.823,-121.698,169.328,48.769,159.279
C04878=1023.026,219.036,-121.721,169.331,48.765,159.278
C04879=1023.031,219.248,-121.743,169.334,48.762,159.278
C04880=1023.036,219.460,-121.766,169.336,48.758,159.278
C04881=1023.041,219.674,-121.789,169.339,48.755,159.277
C04882=1023.047,219.886,-121.812,169.343,48.751,159.277
C04883=1023.052,220.099,-121.834,169.346,48.748,159.277
C04884=1023.058,220.311,-121.857,169.349,48.744,159.276
C04885=1023.063,220.524,-121.880,169.352,48.741,159.276
C04886=1023.069,220.773,-121.906,169.355,48.736,159.276
C04887=1023.076,221.021,-121.934,169.359,48.732,159.275
C04888=1023.082,221.269,-121.960,169.362,48.728,159.275
C04889=1023.089,221.518,-121.987,169.365,48.724,159.274
C04890=1023.095,221.766,-122.013,169.369,48.719,159.274
C04891=1023.101,222.016,-122.040,169.373,48.715,159.274
C04892=1023.108,222.264,-122.066,169.376,48.711,159.273
C04893=1023.113,222.512,-122.093,169.379,48.707,159.273
C04894=1023.120,222.761,-122.120,169.383,48.703,159.273
C04895=1023.126,223.009,-122.146,169.386,48.699,159.272
C04896=1023.133,223.258,-122.173,169.390,48.695,159.272
C04897=1023.139,223.506,-122.201,169.394,48.691,159.272
C04898=1023.146,223.755,-122.227,169.396,48.687,159.271
C04899=1023.152,224.003,-122.254,169.400,48.683,159.271
C04900=1023.158,224.252,-122.281,169.404,48.679,159.271
C04901=1023.164,224.500,-122.307,169.408,48.675,159.270
C04902=1023.171,224.748,-122.334,169.411,48.671,159.270
C04903=1023.177,224.997,-122.361,169.415,48.667,159.270
C04904=1023.184,225.246,-122.388,169.418,48.663,159.269
C04905=1023.190,225.495,-122.415,169.422,48.659,159.269
C04906=1023.197,225.743,-122.441,169.425,48.655,159.268
C04907=1023.204,225.991,-122.468,169.429,48.650,159.268
C04908=1023.209,226.240,-122.495,169.433,48.646,159.268
C04909=1023.216,226.488,-122.521,169.436,48.642,159.267
C04910=1023.222,226.737,-122.548,169.439,48.638,159.267
C04911=1023.229,226.985,-122.576,169.443,48.635,159.267
C04912=1023.235,227.233,-122.602,169.447,48.631,159.266
C04913=1023.241,227.482,-122.630,169.450,48.627,159.266
C04914=1023.248,227.730,-122.656,169.454,48.622,159.266
C04915=1023.254,227.979,-122.683,169.457,48.619,159.265
C04916=1023.261,228.227,-122.711,169.461,48.615,159.265
C04917=1023.267,228.476,-122.738,169.465,48.611,159.265
C04918=1023.273,228.724,-122.765,169.468,48.607,159.264
C04919=1023.279,228.973,-122.792,169.471,48.604,159.264
C04920=1023.286,229.221,-122.820,169.475,48.600,159.264
C04921=1023.292,229.469,-122.846,169.479,48.595,159.263
C04922=1023.298,229.718,-122.874,169.482,48.591,159.263
C04923=1023.305,229.967,-122.901,169.486,48.588,159.263
C04924=1023.310,230.215,-122.928,169.489,48.584,159.263
C04925=1023.318,230.463,-122.955,169.493,48.580,159.262
C04926=1023.324,230.712,-122.983,169.497,48.576,159.262
C04927=1023.330,230.960,-123.010,169.501,48.572,159.262
C04928=1023.336,231.209,-123.038,169.504,48.569,159.261
C04929=1023.342,231.457,-123.064,169.507,48.565,159.261
C04930=1023.349,231.706,-123.092,169.511,48.561,159.261
C04931=1023.355,231.954,-123.120,169.515,48.557,159.261
C04932=1023.361,232.203,-123.146,169.519,48.553,159.260
C04933=1023.368,232.451,-123.174,169.522,48.550,159.260
C04934=1023.375,232.699,-123.202,169.526,48.546,159.260
C04935=1023.380,232.948,-123.228,169.530,48.542,159.259
C04936=1023.387,233.196,-123.256,169.533,48.538,159.259
C04937=1023.394,233.445,-123.284,169.536,48.535,159.259
C04938=1023.403,233.862,-123.330,169.542,48.529,159.258
C04939=1023.414,234.279,-123.376,169.548,48.523,159.258
C04940=1023.426,234.697,-123.422,169.555,48.516,159.257
C04941=1023.435,235.114,-123.468,169.561,48.510,159.257
C04942=1023.442,235.363,-123.496,169.565,48.506,159.257
C04943=1023.449,235.611,-123.524,169.568,48.502,159.256
C04944=1023.455,235.860,-123.550,169.572,48.499,159.256
C04945=1023.461,236.108,-123.578,169.576,48.495,159.256
C04946=1023.468,236.356,-123.606,169.579,48.492,159.256
C04947=1023.475,236.605,-123.634,169.583,48.487,159.255
C04948=1023.481,236.853,-123.661,169.587,48.484,159.255
C04949=1023.487,237.101,-123.689,169.591,48.480,159.255
C04950=1023.494,237.350,-123.716,169.594,48.477,159.254
C04951=1023.500,237.599,-123.744,169.598,48.473,159.254
C04952=1023.506,237.847,-123.771,169.601,48.469,159.254
C04953=1023.512,238.095,-123.799,169.605,48.466,159.254
C04954=1023.519,238.344,-123.827,169.610,48.462,159.254
C04955=1023.526,238.592,-123.855,169.612,48.458,159.253
C04956=1023.532,238.840,-123.882,169.616,48.455,159.253
C04957=1023.538,239.088,-123.910,169.620,48.451,159.253
C04958=1023.544,239.337,-123.938,169.624,48.447,159.252
C04959=1023.551,239.585,-123.966,169.628,48.444,159.252
C04960=1023.558,239.834,-123.993,169.631,48.441,159.252
C04961=1023.564,240.083,-124.022,169.635,48.437,159.252
C04962=1023.570,240.330,-124.049,169.639,48.433,159.251
C04963=1023.577,240.579,-124.077,169.642,48.430,159.251
C04964=1023.582,240.827,-124.105,169.646,48.427,159.251
C04965=1023.589,241.076,-124.133,169.650,48.423,159.251
C04966=1023.595,241.325,-124.161,169.654,48.420,159.251
C04967=1023.602,241.572,-124.190,169.657,48.417,159.250
C04968=1023.608,241.820,-124.217,169.661,48.412,159.250
C04969=1023.614,242.069,-124.245,169.665,48.409,159.250
C04970=1023.621,242.317,-124.273,169.669,48.405,159.250
C04971=1023.627,242.566,-124.301,169.672,48.402,159.250
C04972=1023.633,242.815,-124.329,169.676,48.399,159.249
C04973=1023.640,243.062,-124.358,169.680,48.395,159.249
C04974=1023.646,243.310,-124.386,169.684,48.392,159.249
C04975=1023.652,243.559,-124.413,169.687,48.389,159.249
C04976=1023.658,243.808,-124.442,169.691,48.385,159.248
C04977=1023.665,244.055,-124.470,169.695,48.382,159.248
C04978=1023.671,244.304,-124.498,169.699,48.379,159.248
C04979=1023.678,244.552,-124.527,169.702,48.375,159.248
C04980=1023.684,244.801,-124.556,169.706,48.372,159.248
C04981=1023.690,245.049,-124.583,169.710,48.368,159.248
C04982=1023.696,245.297,-124.612,169.714,48.365,159.247
C04983=1023.702,245.546,-124.640,169.718,48.362,159.247
C04984=1023.709,245.794,-124.669,169.722,48.358,159.247
C04985=1023.715,246.042,-124.697,169.726,48.355,159.247
C04986=1023.721,246.290,-124.726,169.729,48.352,159.247
C04987=1023.728,246.539,-124.754,169.733,48.348,159.246
C04988=1023.734,246.788,-124.782,169.737,48.345,159.246
C04989=1023.740,247.036,-124.811,169.740,48.342,159.246
C04990=1023.747,247.284,-124.839,169.744,48.339,159.246
C04991=1023.753,247.532,-124.868,169.748,48.336,159.246
C04992=1023.759,247.781,-124.896,169.752,48.332,159.246
C04993=1023.765,248.029,-124.925,169.755,48.329,159.245
C04994=1023.775,248.440,-124.973,169.762,48.323,159.245
C04995=1023.786,248.851,-125.020,169.769,48.318,159.245
C04996=1023.796,249.262,-125.067,169.775,48.313,159.245
C04997=1023.807,249.674,-125.114,169.781,48.307,159.244
C04998=1023.814,249.922,-125.143,169.785,48.305,159.244
C04999=1023.820,250.171,-125.171,169.789,48.301,159.244
C05000=1023.827,250.418,-125.200,169.793,48.298,159.244
C05001=1023.833,250.667,-125.229,169.797,48.294,159.244
C05002=1023.839,250.915,-125.257,169.800,48.291,159.243
C05003=1023.845,251.163,-125.286,169.804,48.288,159.243
C05004=1023.852,251.411,-125.315,169.808,48.285,159.243
C05005=1023.858,251.660,-125.343,169.813,48.282,159.243
C05006=1023.864,251.908,-125.372,169.816,48.279,159.243
C05007=1023.871,252.156,-125.400,169.820,48.276,159.243
C05008=1023.877,252.405,-125.429,169.824,48.272,159.243
C05009=1023.883,252.653,-125.458,169.828,48.269,159.243
C05010=1023.890,252.901,-125.487,169.831,48.266,159.242
C05011=1023.897,253.149,-125.515,169.835,48.263,159.242
C05012=1023.903,253.398,-125.544,169.840,48.259,159.242
C05013=1023.909,253.646,-125.573,169.844,48.257,159.242
C05014=1023.916,253.894,-125.601,169.847,48.254,159.242
C05015=1023.923,254.142,-125.631,169.851,48.250,159.242
C05016=1023.929,254.391,-125.659,169.855,48.247,159.242
C05017=1023.935,254.639,-125.688,169.859,48.244,159.242
C05018=1023.942,254.887,-125.716,169.864,48.240,159.241
C05019=1023.948,255.135,-125.745,169.867,48.238,159.241
C05020=1023.955,255.384,-125.775,169.871,48.235,159.241
C05021=1023.962,255.632,-125.803,169.875,48.231,159.241
C05022=1023.968,255.880,-125.832,169.879,48.228,159.241
C05023=1023.974,256.129,-125.861,169.882,48.225,159.241
C05024=1023.980,256.377,-125.890,169.887,48.222,159.241
C05025=1023.988,256.625,-125.918,169.891,48.219,159.240
C05026=1023.994,256.874,-125.947,169.895,48.216,159.240
C05027=1024.000,257.122,-125.977,169.899,48.213,159.240
C05028=1024.007,257.370,-126.006,169.902,48.210,159.240
C05029=1024.014,257.618,-126.034,169.907,48.207,159.240
C05030=1024.021,257.866,-126.063,169.911,48.204,159.240
C05031=1024.027,258.115,-126.092,169.915,48.201,159.240
C05032=1024.033,258.363,-126.121,169.919,48.197,159.240
C05033=1024.040,258.611,-126.150,169.923,48.195,159.240
C05034=1024.047,258.859,-126.179,169.927,48.191,159.239
C05035=1024.053,259.107,-126.208,169.931,48.189,159.239
C05036=1024.060,259.355,-126.237,169.935,48.185,159.239
C05037=1024.067,259.604,-126.266,169.940,48.182,159.239
C05038=1024.073,259.852,-126.295,169.943,48.179,159.239
C05039=1024.079,260.100,-126.324,169.947,48.177,159.239
C05040=1024.086,260.348,-126.353,169.951,48.173,159.239
C05041=1024.093,260.597,-126.382,169.955,48.170,159.239
C05042=1024.100,260.845,-126.412,169.960,48.168,159.239
C05043=1024.106,261.093,-126.441,169.963,48.164,159.239
C05044=1024.112,261.341,-126.471,169.967,48.162,159.239
C05045=1024.119,261.589,-126.501,169.972,48.159,159.239
C05046=1024.125,261.837,-126.530,169.976,48.156,159.239
C05047=1024.131,262.086,-126.559,169.979,48.153,159.238
C05048=1024.138,262.333,-126.589,169.984,48.150,159.238
C05049=1024.145,262.582,-126.618,169.988,48.148,159.238
C05050=1024.155,262.992,-126.667,169.995,48.143,159.238
C05051=1024.165,263.401,-126.715,170.001,48.139,159.238
C05052=1024.176,263.811,-126.764,170.008,48.134,159.238
C05053=1024.187,264.221,-126.813,170.014,48.129,159.238
C05054=1024.193,264.468,-126.842,170.019,48.126,159.238
C05055=1024.200,264.717,-126.872,170.023,48.123,159.238
C05056=1024.207,264.964,-126.902,170.027,48.120,159.238
C05057=1024.212,265.213,-126.931,170.031,48.118,159.238
C05058=1024.219,265.461,-126.961,170.035,48.115,159.238
C05059=1024.226,265.709,-126.990,170.040,48.112,159.238
C05060=1024.232,265.957,-127.020,170.044,48.110,159.238
C05061=1024.239,266.206,-127.050,170.047,48.107,159.238
C05062=1024.245,266.453,-127.080,170.051,48.104,159.238
C05063=1024.252,266.702,-127.110,170.056,48.101,159.238
C05064=1024.258,266.950,-127.139,170.060,48.098,159.238
C05065=1024.264,267.198,-127.169,170.064,48.096,159.237
C05066=1024.271,267.446,-127.199,170.068,48.093,159.237
C05067=1024.278,267.694,-127.229,170.072,48.090,159.237
C05068=1024.285,267.942,-127.259,170.077,48.088,159.237
C05069=1024.290,268.191,-127.288,170.081,48.085,159.237
C05070=1024.297,268.439,-127.318,170.085,48.082,159.237
C05071=1024.304,268.686,-127.348,170.089,48.080,159.237
C05072=1024.310,268.935,-127.378,170.094,48.077,159.238
C05073=1024.317,269.183,-127.408,170.098,48.075,159.238
C05074=1024.323,269.430,-127.438,170.101,48.072,159.237
C05075=1024.330,269.679,-127.468,170.106,48.069,159.237
C05076=1024.336,269.927,-127.497,170.110,48.067,159.237
C05077=1024.343,270.175,-127.528,170.115,48.064,159.237
C05078=1024.349,270.423,-127.558,170.119,48.061,159.237
C05079=1024.356,270.671,-127.588,170.122,48.059,159.237
C05080=1024.362,270.919,-127.618,170.127,48.057,159.238
C05081=1024.369,271.167,-127.649,170.132,48.054,159.238
C05082=1024.375,271.415,-127.679,170.136,48.051,159.238
C05083=1024.382,271.663,-127.709,170.139,48.049,159.238
C05084=1024.388,271.911,-127.739,170.144,48.046,159.237
C05085=1024.395,272.160,-127.769,170.148,48.044,159.238
C05086=1024.401,272.409,-127.799,170.153,48.041,159.238
C05087=1024.408,272.656,-127.829,170.157,48.038,159.238
C05088=1024.414,272.905,-127.860,170.161,48.036,159.238
C05089=1024.421,273.152,-127.890,170.165,48.034,159.238
C05090=1024.427,273.401,-127.920,170.170,48.031,159.238
C05091=1024.434,273.648,-127.950,170.174,48.028,159.238
C05092=1024.440,273.897,-127.981,170.178,48.026,159.238
C05093=1024.446,274.144,-128.012,170.182,48.024,159.238
C05094=1024.453,274.392,-128.042,170.187,48.021,159.238
C05095=1024.460,274.641,-128.073,170.191,48.019,159.238
C05096=1024.466,274.888,-128.103,170.196,48.016,159.238
C05097=1024.473,275.137,-128.133,170.199,48.014,159.238
C05098=1024.480,275.385,-128.163,170.204,48.012,159.238
C05099=1024.486,275.633,-128.194,170.208,48.009,159.238
C05100=1024.492,275.881,-128.224,170.213,48.006,159.238
C05101=1024.499,276.128,-128.255,170.217,48.004,159.238
C05102=1024.505,276.377,-128.286,170.221,48.001,159.238
C05103=1024.512,276.625,-128.316,170.225,47.999,159.238
C05104=1024.518,276.873,-128.346,170.230,47.997,159.238
C05105=1024.525,277.121,-128.376,170.234,47.994,159.238
C05106=1024.536,277.535,-128.428,170.242,47.990,159.239
C05107=1024.547,277.949,-128.480,170.249,47.987,159.239
C05108=1024.558,278.363,-128.531,170.256,47.982,159.239
C05109=1024.569,278.778,-128.582,170.264,47.979,159.239
C05110=1024.574,279.026,-128.613,170.268,47.976,159.239
C05111=1024.582,279.274,-128.644,170.272,47.974,159.239
C05112=1024.588,279.522,-128.674,170.276,47.972,159.239
C05113=1024.594,279.769,-128.705,170.281,47.969,159.239
C05114=1024.601,280.018,-128.736,170.286,47.967,159.240
C05115=1024.608,280.266,-128.768,170.290,47.965,159.240
C05116=1024.614,280.514,-128.798,170.294,47.963,159.240
C05117=1024.621,280.761,-128.829,170.298,47.961,159.240
C05118=1024.627,281.010,-128.860,170.303,47.958,159.240
C05119=1024.634,281.257,-128.891,170.307,47.956,159.240
C05120=1024.640,281.506,-128.922,170.312,47.954,159.240
C05121=1024.647,281.754,-128.953,170.316,47.952,159.240
C05122=1024.653,282.002,-128.983,170.320,47.949,159.240
C05123=1024.660,282.249,-129.014,170.325,47.947,159.240
C05124=1024.667,282.497,-129.046,170.330,47.945,159.241
C05125=1024.674,282.746,-129.076,170.334,47.943,159.241
C05126=1024.680,282.994,-129.108,170.339,47.940,159.241
C05127=1024.686,283.241,-129.138,170.343,47.938,159.241
C05128=1024.693,283.489,-129.170,170.347,47.936,159.241
C05129=1024.700,283.737,-129.201,170.352,47.934,159.241
C05130=1024.707,283.986,-129.231,170.356,47.931,159.241
C05131=1024.713,284.233,-129.263,170.361,47.929,159.241
C05132=1024.720,284.481,-129.294,170.366,47.927,159.242
C05133=1024.727,284.729,-129.326,170.370,47.925,159.242
C05134=1024.733,284.977,-129.356,170.374,47.923,159.242
C05135=1024.739,285.225,-129.387,170.379,47.921,159.242
C05136=1024.747,285.473,-129.418,170.383,47.918,159.242
C05137=1024.754,285.720,-129.450,170.388,47.916,159.242
C05138=1024.760,285.969,-129.482,170.393,47.914,159.242
C05139=1024.766,286.217,-129.512,170.398,47.912,159.243
C05140=1024.773,286.465,-129.544,170.401,47.910,159.243
C05141=1024.779,286.713,-129.575,170.406,47.908,159.243
C05142=1024.786,286.961,-129.607,170.411,47.906,159.243
C05143=1024.793,287.209,-129.638,170.415,47.904,159.243
C05144=1024.800,287.457,-129.669,170.420,47.902,159.243
C05145=1024.806,287.704,-129.701,170.425,47.900,159.243
C05146=1024.813,287.952,-129.732,170.429,47.898,159.244
C05147=1024.819,288.200,-129.763,170.433,47.896,159.244
C05148=1024.826,288.448,-129.795,170.438,47.894,159.244
C05149=1024.833,288.695,-129.826,170.443,47.892,159.244
C05150=1024.839,288.944,-129.858,170.447,47.890,159.244
C05151=1024.845,289.192,-129.890,170.452,47.888,159.244
C05152=1024.852,289.440,-129.921,170.457,47.886,159.245
C05153=1024.859,289.687,-129.953,170.461,47.884,159.245
C05154=1024.866,289.935,-129.985,170.466,47.882,159.245
C05155=1024.873,290.183,-130.016,170.470,47.880,159.245
C05156=1024.879,290.431,-130.048,170.475,47.878,159.245
C05157=1024.885,290.679,-130.080,170.480,47.876,159.246
C05158=1024.892,290.927,-130.111,170.484,47.874,159.246
C05159=1024.899,291.174,-130.143,170.490,47.872,159.246
C05160=1024.906,291.422,-130.175,170.494,47.870,159.246
C05161=1024.913,291.670,-130.206,170.498,47.869,159.246
C05162=1024.918,291.884,-130.234,170.503,47.866,159.247
C05163=1024.924,292.097,-130.261,170.507,47.865,159.247
C05164=1024.930,292.309,-130.288,170.510,47.863,159.247
C05165=1024.935,292.523,-130.316,170.514,47.862,159.247
C05166=1024.942,292.736,-130.344,170.518,47.861,159.247
C05167=1024.947,292.950,-130.370,170.523,47.858,159.248
C05168=1024.953,293.163,-130.398,170.527,47.857,159.248
C05169=1024.959,293.376,-130.426,170.531,47.855,159.248
C05170=1024.965,293.624,-130.458,170.535,47.853,159.248
C05171=1024.972,293.872,-130.489,170.540,47.852,159.248
C05172=1024.979,294.119,-130.522,170.545,47.850,159.249
C05173=1024.985,294.367,-130.554,170.550,47.848,159.249
C05174=1024.991,294.615,-130.586,170.554,47.847,159.249
C05175=1024.998,294.862,-130.618,170.559,47.845,159.249
C05176=1025.004,295.111,-130.650,170.564,47.843,159.250
C05177=1025.011,295.358,-130.683,170.569,47.842,159.250
C05178=1025.018,295.606,-130.715,170.573,47.840,159.250
C05179=1025.024,295.854,-130.748,170.578,47.838,159.250
C05180=1025.031,296.102,-130.780,170.583,47.836,159.251
C05181=1025.037,296.349,-130.813,170.587,47.835,159.251
C05182=1025.043,296.598,-130.845,170.592,47.833,159.251
C05183=1025.050,296.845,-130.877,170.597,47.831,159.251
C05184=1025.057,297.092,-130.910,170.602,47.830,159.252
C05185=1025.063,297.341,-130.942,170.607,47.828,159.252
C05186=1025.070,297.589,-130.974,170.612,47.826,159.252
C05187=1025.077,297.836,-131.007,170.616,47.824,159.252
C05188=1025.084,298.083,-131.039,170.622,47.823,159.253
C05189=1025.090,298.331,-131.072,170.626,47.822,159.253
C05190=1025.097,298.580,-131.104,170.630,47.820,159.253
C05191=1025.104,298.827,-131.136,170.635,47.818,159.254
C05192=1025.110,299.075,-131.169,170.640,47.817,159.254
C05193=1025.116,299.322,-131.202,170.645,47.815,159.254
C05194=1025.124,299.570,-131.234,170.650,47.813,159.255
C05195=1025.130,299.818,-131.267,170.655,47.812,159.255
C05196=1025.136,300.066,-131.300,170.660,47.810,159.255
C05197=1025.143,300.314,-131.331,170.665,47.808,159.255
C05198=1025.150,300.562,-131.364,170.670,47.807,159.256
C05199=1025.157,300.809,-131.396,170.675,47.805,159.256
C05200=1025.163,301.057,-131.429,170.680,47.803,159.256
C05201=1025.170,301.305,-131.462,170.685,47.802,159.257
C05202=1025.177,301.552,-131.494,170.689,47.801,159.257
C05203=1025.184,301.800,-131.527,170.694,47.799,159.257
C05204=1025.190,302.048,-131.560,170.699,47.798,159.258
C05205=1025.198,302.295,-131.592,170.704,47.796,159.258
C05206=1025.204,302.544,-131.626,170.709,47.794,159.258
C05207=1025.211,302.791,-131.658,170.714,47.793,159.258
C05208=1025.218,303.038,-131.691,170.719,47.791,159.259
C05209=1025.225,303.286,-131.724,170.724,47.790,159.259
C05210=1025.231,303.534,-131.757,170.729,47.788,159.260
C05211=1025.239,303.782,-131.790,170.734,47.787,159.260
C05212=1025.245,304.029,-131.822,170.739,47.785,159.260
C05213=1025.252,304.278,-131.855,170.744,47.783,159.260
C05214=1025.259,304.525,-131.888,170.749,47.782,159.261
C05215=1025.266,304.772,-131.921,170.754,47.780,159.261
C05216=1025.273,305.020,-131.954,170.759,47.779,159.261
C05217=1025.280,305.268,-131.986,170.764,47.778,159.262
C05218=1025.287,305.516,-132.019,170.769,47.776,159.262
C05219=1025.293,305.763,-132.052,170.774,47.775,159.263
C05220=1025.301,306.011,-132.085,170.779,47.773,159.263
C05221=1025.307,306.258,-132.118,170.784,47.772,159.263
C05222=1025.314,306.481,-132.148,170.789,47.770,159.264
C05223=1025.320,306.702,-132.177,170.793,47.769,159.264
C05224=1025.326,306.924,-132.207,170.798,47.768,159.264
C05225=1025.332,307.146,-132.236,170.802,47.767,159.264
C05226=1025.339,307.368,-132.266,170.807,47.765,159.265
C05227=1025.345,307.590,-132.295,170.811,47.764,159.265
C05228=1025.351,307.812,-132.325,170.816,47.762,159.265
C05229=1025.357,308.033,-132.355,170.820,47.761,159.266
C05230=1025.364,308.281,-132.388,170.826,47.760,159.266
C05231=1025.372,308.529,-132.421,170.831,47.759,159.267
C05232=1025.378,308.776,-132.454,170.836,47.758,159.267
C05233=1025.386,309.024,-132.488,170.841,47.756,159.267
C05234=1025.393,309.272,-132.520,170.846,47.755,159.268
C05235=1025.400,309.519,-132.554,170.852,47.753,159.268
C05236=1025.407,309.767,-132.587,170.857,47.752,159.268
C05237=1025.415,310.015,-132.620,170.862,47.750,159.269
C05238=1025.421,310.262,-132.653,170.867,47.749,159.269
C05239=1025.428,310.510,-132.686,170.872,47.748,159.270
C05240=1025.435,310.757,-132.720,170.877,47.746,159.270
C05241=1025.442,311.005,-132.753,170.883,47.746,159.271
C05242=1025.449,311.253,-132.787,170.888,47.744,159.271
C05243=1025.455,311.500,-132.821,170.893,47.743,159.271
C05244=1025.462,311.748,-132.855,170.898,47.742,159.272
C05245=1025.469,311.996,-132.889,170.903,47.741,159.272
C05246=1025.475,312.243,-132.923,170.908,47.740,159.273
C05247=1025.482,312.491,-132.956,170.914,47.739,159.273
C05248=1025.489,312.738,-132.990,170.919,47.737,159.274
C05249=1025.496,312.985,-133.024,170.924,47.736,159.274
C05250=1025.502,313.233,-133.058,170.929,47.735,159.274
C05251=1025.510,313.481,-133.092,170.935,47.734,159.275
C05252=1025.516,313.728,-133.125,170.940,47.733,159.275
C05253=1025.523,313.976,-133.160,170.945,47.732,159.276
C05254=1025.530,314.223,-133.194,170.950,47.731,159.276
C05255=1025.537,314.471,-133.227,170.955,47.730,159.277
C05256=1025.543,314.718,-133.261,170.961,47.729,159.277
C05257=1025.550,314.966,-133.295,170.966,47.727,159.278
C05258=1025.557,315.214,-133.329,170.971,47.727,159.278
C05259=1025.564,315.461,-133.363,170.976,47.726,159.279
C05260=1025.570,315.709,-133.397,170.982,47.724,159.279
C05261=1025.578,315.956,-133.431,170.987,47.724,159.280
C05262=1025.585,316.204,-133.465,170.993,47.722,159.280
C05263=1025.592,316.451,-133.500,170.998,47.721,159.280
C05264=1025.599,316.699,-133.534,171.004,47.720,159.281
C05265=1025.606,316.947,-133.567,171.009,47.719,159.282
C05266=1025.612,317.195,-133.602,171.014,47.719,159.282
C05267=1025.619,317.441,-133.636,171.019,47.717,159.282
C05268=1025.626,317.689,-133.670,171.025,47.716,159.283
C05269=1025.633,317.937,-133.704,171.030,47.715,159.283
C05270=1025.640,318.184,-133.738,171.035,47.715,159.284
C05271=1025.648,318.431,-133.773,171.041,47.713,159.284
C05272=1025.654,318.679,-133.807,171.047,47.712,159.285
C05273=1025.661,318.927,-133.841,171.052,47.711,159.285
C05274=1025.669,319.174,-133.875,171.058,47.710,159.286
C05275=1025.675,319.422,-133.910,171.063,47.710,159.287
C05276=1025.682,319.670,-133.944,171.068,47.709,159.287
C05277=1025.690,319.917,-133.978,171.074,47.708,159.288
C05278=1025.696,320.165,-134.013,171.079,47.707,159.288
C05279=1025.704,320.412,-134.047,171.085,47.705,159.289
C05280=1025.711,320.660,-134.081,171.090,47.705,159.289
C05281=1025.718,320.907,-134.116,171.096,47.704,159.290
C05282=1025.725,321.131,-134.147,171.101,47.703,159.290
C05283=1025.731,321.356,-134.178,171.105,47.702,159.291
C05284=1025.737,321.580,-134.209,171.111,47.702,159.291
C05285=1025.744,321.804,-134.241,171.116,47.701,159.292
C05286=1025.750,322.029,-134.272,171.121,47.700,159.292
C05287=1025.756,322.253,-134.303,171.126,47.699,159.293
C05288=1025.763,322.478,-134.334,171.131,47.698,159.293
C05289=1025.770,322.703,-134.366,171.136,47.697,159.294
C05290=1025.778,322.950,-134.401,171.142,47.696,159.294
C05291=1025.784,323.198,-134.435,171.147,47.696,159.295
C05292=1025.792,323.445,-134.469,171.153,47.695,159.295
C05293=1025.799,323.692,-134.504,171.158,47.695,159.296
C05294=1025.806,323.940,-134.538,171.164,47.693,159.296
C05295=1025.814,324.188,-134.573,171.170,47.693,159.297
C05296=1025.821,324.435,-134.608,171.175,47.692,159.297
C05297=1025.828,324.682,-134.643,171.180,47.691,159.298
C05298=1025.835,324.930,-134.677,171.187,47.690,159.299
C05299=1025.843,325.177,-134.711,171.192,47.689,159.299
C05300=1025.850,325.425,-134.747,171.198,47.689,159.300
C05301=1025.858,325.672,-134.781,171.203,47.688,159.300
C05302=1025.864,325.920,-134.816,171.210,47.687,159.301
C05303=1025.872,326.168,-134.851,171.215,47.686,159.301
C05304=1025.880,326.415,-134.885,171.220,47.685,159.302
C05305=1025.886,326.662,-134.920,171.226,47.685,159.303
C05306=1025.894,326.909,-134.955,171.232,47.684,159.303
C05307=1025.902,327.157,-134.990,171.238,47.683,159.304
C05308=1025.909,327.404,-135.025,171.243,47.683,159.305
C05309=1025.916,327.652,-135.060,171.249,47.682,159.305
C05310=1025.923,327.900,-135.096,171.255,47.682,159.306
C05311=1025.930,328.147,-135.130,171.261,47.681,159.306
C05312=1025.937,328.393,-135.166,171.266,47.680,159.307
C05313=1025.945,328.641,-135.202,171.272,47.680,159.308
C05314=1025.952,328.889,-135.237,171.278,47.679,159.308
C05315=1025.958,329.136,-135.272,171.284,47.678,159.309
C05316=1025.967,329.384,-135.307,171.290,47.678,159.310
C05317=1025.974,329.631,-135.343,171.295,47.677,159.310
C05318=1025.980,329.878,-135.378,171.302,47.677,159.311
C05319=1025.988,330.126,-135.413,171.307,47.676,159.312
C05320=1025.995,330.373,-135.449,171.313,47.676,159.312
C05321=1026.003,330.621,-135.484,171.319,47.675,159.313
C05322=1026.010,330.868,-135.519,171.325,47.675,159.314
C05323=1026.017,331.115,-135.555,171.330,47.674,159.314
C05324=1026.024,331.363,-135.590,171.336,47.674,159.315
C05325=1026.031,331.610,-135.626,171.342,47.673,159.316
C05326=1026.039,331.857,-135.661,171.348,47.673,159.316
C05327=1026.046,332.105,-135.696,171.354,47.673,159.317
C05328=1026.054,332.352,-135.733,171.360,47.672,159.318
C05329=1026.061,332.600,-135.768,171.366,47.671,159.318
C05330=1026.068,332.847,-135.804,171.371,47.671,159.319
C05331=1026.075,333.094,-135.839,171.378,47.671,159.320
C05332=1026.083,333.341,-135.875,171.383,47.670,159.320
C05333=1026.090,333.588,-135.910,171.389,47.670,159.321
C05334=1026.098,333.836,-135.946,171.396,47.669,159.322
C05335=1026.105,334.084,-135.982,171.401,47.669,159.323
C05336=1026.113,334.330,-136.018,171.407,47.669,159.323
C05337=1026.120,334.579,-136.054,171.414,47.668,159.324
C05338=1026.126,334.826,-136.090,171.420,47.668,159.325
C05339=1026.134,335.073,-136.126,171.425,47.668,159.325
C05340=1026.141,335.320,-136.162,171.432,47.667,159.326
C05341=1026.149,335.567,-136.198,171.438,47.667,159.327
C05342=1026.155,335.790,-136.230,171.443,47.666,159.327
C05343=1026.162,336.012,-136.263,171.449,47.666,159.328
C05344=1026.169,336.234,-136.295,171.454,47.666,159.329
C05345=1026.175,336.456,-136.328,171.459,47.666,159.330
C05346=1026.182,336.679,-136.359,171.465,47.666,159.330
C05347=1026.188,336.901,-136.392,171.470,47.666,159.331
C05348=1026.195,337.123,-136.424,171.476,47.665,159.331
C05349=1026.202,337.345,-136.457,171.481,47.665,159.332
C05350=1026.209,337.592,-136.493,171.487,47.664,159.333
C05351=1026.217,337.839,-136.529,171.494,47.664,159.334
C05352=1026.224,338.087,-136.565,171.500,47.664,159.335
C05353=1026.232,338.334,-136.602,171.505,47.664,159.335
C05354=1026.239,338.581,-136.637,171.512,47.663,159.336
C05355=1026.247,338.828,-136.674,171.518,47.663,159.337
C05356=1026.254,339.076,-136.710,171.525,47.663,159.338
C05357=1026.261,339.323,-136.747,171.530,47.663,159.338
C05358=1026.269,339.570,-136.784,171.537,47.663,159.339
C05359=1026.276,339.817,-136.819,171.543,47.662,159.340
C05360=1026.284,340.064,-136.856,171.550,47.663,159.341
